C09106=1039.782,271.564,387.906,171.420,41.865,158.001
C09107=1039.788,271.812,387.876,171.423,41.867,158.001
C09108=1039.795,272.060,387.845,171.427,41.868,158.002
C09109=1039.802,272.308,387.814,171.430,41.870,158.002
C09110=1039.809,272.556,387.784,171.433,41.871,158.003
C09111=1039.815,272.805,387.753,171.437,41.873,158.003
C09112=1039.821,273.052,387.722,171.439,41.875,158.004
C09113=1039.828,273.300,387.692,171.443,41.876,158.004
C09114=1039.835,273.548,387.660,171.447,41.878,158.005
C09115=1039.842,273.796,387.630,171.449,41.880,158.006
C09116=1039.849,274.044,387.599,171.453,41.881,158.006
C09117=1039.855,274.292,387.568,171.457,41.883,158.007
C09118=1039.862,274.540,387.538,171.459,41.885,158.007
C09119=1039.869,274.788,387.507,171.463,41.887,158.008
C09120=1039.876,275.036,387.475,171.466,41.888,158.009
C09121=1039.882,275.285,387.445,171.469,41.890,158.009
C09122=1039.889,275.532,387.414,171.473,41.892,158.010
C09123=1039.895,275.780,387.383,171.475,41.893,158.010
C09124=1039.902,276.028,387.352,171.479,41.895,158.011
C09125=1039.908,276.276,387.321,171.483,41.897,158.011
C09126=1039.916,276.524,387.290,171.485,41.898,158.012
C09127=1039.925,276.838,387.251,171.490,41.901,158.013
C09128=1039.933,277.151,387.212,171.494,41.903,158.013
C09129=1039.942,277.465,387.173,171.498,41.905,158.014
C09130=1039.950,277.778,387.133,171.503,41.907,158.015
C09131=1039.957,278.027,387.103,171.507,41.909,158.016
C09132=1039.963,278.274,387.072,171.509,41.910,158.016
C09133=1039.970,278.522,387.040,171.513,41.912,158.017
C09134=1039.977,278.770,387.010,171.516,41.914,158.017
C09135=1039.983,279.018,386.979,171.519,41.916,158.018
C09136=1039.990,279.266,386.947,171.523,41.917,158.018
C09137=1039.997,279.514,386.916,171.527,41.919,158.019
C09138=1040.004,279.762,386.884,171.529,41.921,158.020
C09139=1040.010,280.010,386.854,171.533,41.923,158.020
C09140=1040.017,280.258,386.822,171.537,41.925,158.021
C09141=1040.023,280.506,386.791,171.539,41.926,158.021
C09142=1040.030,280.754,386.759,171.543,41.928,158.022
C09143=1040.037,281.002,386.728,171.547,41.930,158.023
C09144=1040.044,281.250,386.696,171.551,41.932,158.023
C09145=1040.050,281.498,386.665,171.553,41.933,158.024
C09146=1040.057,281.745,386.634,171.557,41.935,158.025
C09147=1040.063,281.993,386.602,171.561,41.937,158.025
C09148=1040.070,282.241,386.571,171.563,41.939,158.026
C09149=1040.077,282.489,386.540,171.567,41.941,158.026
C09150=1040.083,282.736,386.508,171.571,41.942,158.027
C09151=1040.090,282.984,386.477,171.574,41.944,158.028
C09152=1040.097,283.232,386.445,171.577,41.946,158.028
C09153=1040.104,283.481,386.413,171.581,41.948,158.029
C09154=1040.111,283.729,386.382,171.585,41.950,158.029
C09155=1040.118,283.977,386.351,171.588,41.951,158.030
C09156=1040.124,284.225,386.319,171.592,41.953,158.031
C09157=1040.131,284.473,386.288,171.595,41.954,158.031
C09158=1040.138,284.720,386.256,171.598,41.956,158.032
C09159=1040.145,284.968,386.225,171.602,41.958,158.033
C09160=1040.151,285.216,386.193,171.606,41.960,158.033
C09161=1040.158,285.463,386.161,171.608,41.962,158.034
C09162=1040.165,285.711,386.130,171.612,41.964,158.034
C09163=1040.172,285.959,386.098,171.616,41.965,158.035
C09164=1040.178,286.207,386.067,171.620,41.967,158.036
C09165=1040.185,286.455,386.036,171.623,41.969,158.036
C09166=1040.193,286.704,386.004,171.626,41.971,158.037
C09167=1040.200,286.951,385.972,171.630,41.973,158.037
C09168=1040.206,287.199,385.940,171.633,41.974,158.038
C09169=1040.212,287.447,385.908,171.637,41.976,158.039
C09170=1040.219,287.694,385.876,171.641,41.978,158.039
C09171=1040.226,287.942,385.845,171.645,41.980,158.040
C09172=1040.232,288.191,385.813,171.647,41.982,158.041
C09173=1040.239,288.438,385.780,171.651,41.984,158.041
C09174=1040.246,288.686,385.749,171.655,41.986,158.042
C09175=1040.253,288.934,385.717,171.659,41.988,158.043
C09176=1040.260,289.182,385.685,171.662,41.989,158.043
C09177=1040.266,289.430,385.653,171.665,41.991,158.044
C09178=1040.273,289.677,385.621,171.669,41.993,158.044
C09179=1040.280,289.925,385.589,171.673,41.995,158.045
C09180=1040.287,290.173,385.556,171.676,41.997,158.046
C09181=1040.293,290.421,385.525,171.680,41.999,158.046
C09182=1040.301,290.668,385.493,171.684,42.001,158.047
C09183=1040.309,290.994,385.451,171.688,42.003,158.048
C09184=1040.318,291.320,385.408,171.693,42.006,158.049
C09185=1040.327,291.645,385.366,171.698,42.008,158.050
C09186=1040.336,291.971,385.325,171.703,42.011,158.051
C09187=1040.343,292.218,385.292,171.707,42.013,158.051
C09188=1040.349,292.466,385.260,171.710,42.015,158.052
C09189=1040.356,292.714,385.228,171.713,42.017,158.052
C09190=1040.364,292.962,385.196,171.717,42.019,158.053
C09191=1040.370,293.209,385.163,171.721,42.021,158.054
C09192=1040.377,293.457,385.132,171.725,42.023,158.055
C09193=1040.384,293.704,385.099,171.728,42.025,158.055
C09194=1040.391,293.953,385.066,171.732,42.027,158.056
C09195=1040.397,294.201,385.035,171.736,42.029,158.057
C09196=1040.404,294.448,385.002,171.740,42.031,158.057
C09197=1040.411,294.696,384.970,171.743,42.032,158.058
C09198=1040.418,294.944,384.937,171.747,42.034,158.058
C09199=1040.425,295.191,384.905,171.750,42.036,158.059
C09200=1040.431,295.439,384.873,171.754,42.038,158.060
C09201=1040.438,295.687,384.840,171.757,42.040,158.061
C09202=1040.445,295.935,384.807,171.761,42.043,158.061
C09203=1040.451,296.182,384.775,171.765,42.045,158.062
C09204=1040.458,296.431,384.742,171.769,42.047,158.063
C09205=1040.465,296.678,384.709,171.773,42.048,158.063
C09206=1040.471,296.926,384.677,171.777,42.050,158.064
C09207=1040.477,297.173,384.644,171.780,42.052,158.065
C09208=1040.484,297.422,384.611,171.784,42.054,158.065
C09209=1040.491,297.669,384.578,171.788,42.057,158.066
C09210=1040.498,297.916,384.546,171.792,42.059,158.067
C09211=1040.505,298.165,384.513,171.795,42.061,158.068
C09212=1040.511,298.412,384.480,171.799,42.063,158.068
C09213=1040.517,298.660,384.447,171.802,42.065,158.069
C09214=1040.525,298.907,384.414,171.806,42.067,158.070
C09215=1040.531,299.155,384.381,171.810,42.070,158.071
C09216=1040.538,299.402,384.349,171.814,42.072,158.071
C09217=1040.545,299.651,384.315,171.818,42.074,158.072
C09218=1040.551,299.898,384.283,171.822,42.076,158.073
C09219=1040.558,300.146,384.250,171.825,42.077,158.073
C09220=1040.565,300.394,384.217,171.829,42.080,158.074
C09221=1040.571,300.641,384.184,171.833,42.082,158.075
C09222=1040.578,300.889,384.151,171.837,42.084,158.075
C09223=1040.585,301.136,384.119,171.841,42.086,158.076
C09224=1040.592,301.385,384.086,171.845,42.088,158.077
C09225=1040.599,301.632,384.052,171.849,42.091,158.078
C09226=1040.606,301.880,384.019,171.852,42.092,158.078
C09227=1040.612,302.128,383.986,171.856,42.094,158.079
C09228=1040.620,302.375,383.953,171.860,42.096,158.080
C09229=1040.626,302.623,383.920,171.864,42.099,158.081
C09230=1040.633,302.871,383.887,171.868,42.101,158.081
C09231=1040.640,303.118,383.854,171.872,42.103,158.082
C09232=1040.647,303.366,383.821,171.876,42.106,158.083
C09233=1040.653,303.614,383.788,171.879,42.107,158.083
C09234=1040.661,303.861,383.755,171.883,42.109,158.084
C09235=1040.667,304.109,383.722,171.887,42.111,158.085
C09236=1040.674,304.356,383.688,171.891,42.114,158.086
C09237=1040.681,304.604,383.655,171.896,42.116,158.086
C09238=1040.687,304.852,383.622,171.900,42.118,158.087
C09239=1040.697,305.194,383.576,171.905,42.121,158.088
C09240=1040.707,305.536,383.530,171.910,42.124,158.089
C09241=1040.717,305.878,383.485,171.915,42.127,158.090
C09242=1040.726,306.220,383.439,171.921,42.130,158.091
C09243=1040.733,306.467,383.406,171.925,42.132,158.092
C09244=1040.740,306.715,383.372,171.929,42.134,158.093
C09245=1040.747,306.963,383.339,171.933,42.137,158.094
C09246=1040.754,307.210,383.305,171.937,42.139,158.094
C09247=1040.761,307.458,383.272,171.941,42.141,158.095
C09248=1040.769,307.705,383.239,171.945,42.143,158.096
C09249=1040.775,307.953,383.206,171.950,42.145,158.097
C09250=1040.782,308.201,383.172,171.954,42.148,158.097
C09251=1040.789,308.448,383.138,171.957,42.150,158.098
C09252=1040.796,308.695,383.105,171.961,42.151,158.099
C09253=1040.803,308.944,383.072,171.965,42.154,158.100
C09254=1040.810,309.191,383.038,171.969,42.156,158.100
C09255=1040.818,309.439,383.005,171.973,42.159,158.101
C09256=1040.824,309.686,382.972,171.978,42.160,158.102
C09257=1040.831,309.934,382.938,171.982,42.163,158.103
C09258=1040.839,310.182,382.904,171.986,42.165,158.103
C09259=1040.846,310.429,382.871,171.990,42.167,158.104
C09260=1040.852,310.676,382.837,171.993,42.169,158.105
C09261=1040.859,310.925,382.804,171.998,42.172,158.106
C09262=1040.867,311.172,382.770,172.002,42.174,158.106
C09263=1040.874,311.420,382.737,172.006,42.176,158.107
C09264=1040.882,311.667,382.703,172.010,42.178,158.108
C09265=1040.889,311.915,382.669,172.014,42.181,158.109
C09266=1040.895,312.162,382.636,172.019,42.183,158.110
C09267=1040.903,312.410,382.602,172.023,42.185,158.110
C09268=1040.909,312.658,382.568,172.027,42.188,158.111
C09269=1040.916,312.905,382.534,172.031,42.190,158.112
C09270=1040.922,313.152,382.500,172.035,42.192,158.113
C09271=1040.929,313.400,382.466,172.039,42.195,158.114
C09272=1040.936,313.648,382.431,172.044,42.197,158.115
C09273=1040.943,313.895,382.397,172.048,42.200,158.115
C09274=1040.949,314.142,382.363,172.051,42.202,158.116
C09275=1040.956,314.390,382.329,172.055,42.204,158.117
C09276=1040.964,314.638,382.295,172.060,42.207,158.118
C09277=1040.970,314.885,382.260,172.064,42.209,158.119
C09278=1040.978,315.133,382.226,172.069,42.212,158.119
C09279=1040.984,315.381,382.192,172.073,42.214,158.120
C09280=1040.991,315.627,382.158,172.077,42.217,158.121
C09281=1040.997,315.875,382.123,172.080,42.219,158.122
C09282=1041.005,316.123,382.089,172.085,42.221,158.123
C09283=1041.011,316.370,382.054,172.089,42.224,158.124
C09284=1041.019,316.618,382.020,172.093,42.226,158.124
C09285=1041.025,316.866,381.986,172.097,42.229,158.125
C09286=1041.033,317.113,381.952,172.101,42.231,158.126
C09287=1041.039,317.361,381.917,172.106,42.234,158.127
C09288=1041.046,317.609,381.883,172.110,42.236,158.128
C09289=1041.052,317.855,381.849,172.114,42.239,158.129
C09290=1041.060,318.103,381.815,172.119,42.241,158.130
C09291=1041.066,318.350,381.780,172.123,42.244,158.130
C09292=1041.074,318.598,381.746,172.127,42.246,158.131
C09293=1041.080,318.845,381.711,172.132,42.249,158.132
C09294=1041.088,319.093,381.677,172.137,42.251,158.133
C09295=1041.098,319.440,381.628,172.142,42.255,158.134
C09296=1041.107,319.787,381.580,172.148,42.258,158.135
C09297=1041.117,320.133,381.531,172.155,42.261,158.137
C09298=1041.127,320.480,381.483,172.160,42.265,158.138
C09299=1041.134,320.728,381.448,172.164,42.268,158.139
C09300=1041.141,320.975,381.414,172.169,42.270,158.139
C09301=1041.148,321.222,381.378,172.173,42.273,158.140
C09302=1041.155,321.470,381.345,172.177,42.275,158.141
C09303=1041.162,321.717,381.310,172.182,42.277,158.142
C09304=1041.169,321.964,381.275,172.186,42.280,158.143
C09305=1041.177,322.213,381.240,172.191,42.282,158.144
C09306=1041.184,322.460,381.206,172.195,42.285,158.145
C09307=1041.191,322.707,381.171,172.200,42.288,158.146
C09308=1041.198,322.954,381.136,172.205,42.290,158.147
C09309=1041.205,323.202,381.102,172.209,42.293,158.147
C09310=1041.212,323.449,381.067,172.213,42.295,158.148
C09311=1041.220,323.697,381.032,172.218,42.298,158.149
C09312=1041.226,323.945,380.996,172.222,42.300,158.150
C09313=1041.234,324.192,380.962,172.227,42.303,158.151
C09314=1041.241,324.439,380.927,172.231,42.306,158.152
C09315=1041.248,324.686,380.892,172.235,42.308,158.153
C09316=1041.255,324.935,380.857,172.240,42.311,158.154
C09317=1041.263,325.182,380.823,172.244,42.313,158.154
C09318=1041.270,325.429,380.788,172.249,42.316,158.155
C09319=1041.277,325.676,380.753,172.253,42.319,158.156
C09320=1041.284,325.925,380.718,172.257,42.321,158.157
C09321=1041.291,326.172,380.683,172.262,42.324,158.158
C09322=1041.299,326.419,380.648,172.266,42.327,158.159
C09323=1041.306,326.667,380.612,172.272,42.329,158.160
C09324=1041.314,326.914,380.578,172.276,42.332,158.161
C09325=1041.320,327.161,380.543,172.281,42.334,158.162
C09326=1041.328,327.409,380.508,172.285,42.337,158.163
C09327=1041.336,327.656,380.472,172.290,42.339,158.164
C09328=1041.342,327.903,380.437,172.294,42.342,158.164
C09329=1041.350,328.151,380.402,172.299,42.345,158.165
C09330=1041.357,328.398,380.367,172.303,42.347,158.166
C09331=1041.365,328.646,380.332,172.308,42.350,158.167
C09332=1041.372,328.894,380.297,172.312,42.353,158.168
C09333=1041.379,329.140,380.261,172.317,42.355,158.169
C09334=1041.386,329.388,380.225,172.322,42.358,158.170
C09335=1041.393,329.636,380.190,172.327,42.361,158.171
C09336=1041.400,329.882,380.154,172.331,42.364,158.172
C09337=1041.408,330.131,380.119,172.336,42.367,158.173
C09338=1041.414,330.378,380.084,172.340,42.369,158.174
C09339=1041.422,330.625,380.048,172.345,42.372,158.175
C09340=1041.429,330.873,380.013,172.349,42.375,158.176
C09341=1041.436,331.119,379.977,172.355,42.378,158.177
C09342=1041.443,331.368,379.941,172.359,42.381,158.178
C09343=1041.450,331.614,379.905,172.364,42.383,158.179
C09344=1041.458,331.862,379.870,172.368,42.386,158.180
C09345=1041.465,332.109,379.834,172.373,42.389,158.181
C09346=1041.472,332.357,379.798,172.377,42.392,158.182
C09347=1041.479,332.604,379.763,172.383,42.395,158.183
C09348=1041.487,332.852,379.727,172.387,42.398,158.184
C09349=1041.494,333.099,379.691,172.392,42.400,158.185
C09350=1041.501,333.345,379.655,172.396,42.403,158.186
C09351=1041.511,333.688,379.606,172.403,42.407,158.187
C09352=1041.521,334.030,379.556,172.409,42.411,158.188
C09353=1041.531,334.371,379.507,172.416,42.415,158.190
C09354=1041.542,334.714,379.457,172.423,42.419,158.191
C09355=1041.548,334.961,379.422,172.428,42.422,158.192
C09356=1041.556,335.208,379.386,172.432,42.425,158.193
C09357=1041.564,335.456,379.349,172.437,42.428,158.194
C09358=1041.571,335.703,379.313,172.442,42.431,158.195
C09359=1041.578,335.950,379.277,172.447,42.433,158.196
C09360=1041.585,336.197,379.241,172.452,42.436,158.197
C09361=1041.592,336.445,379.205,172.456,42.439,158.198
C09362=1041.599,336.692,379.169,172.461,42.442,158.199
C09363=1041.607,336.939,379.133,172.467,42.445,158.200
C09364=1041.614,337.187,379.096,172.471,42.448,158.201
C09365=1041.621,337.434,379.061,172.476,42.451,158.202
C09366=1041.629,337.681,379.024,172.480,42.454,158.203
C09367=1041.635,337.929,378.988,172.486,42.457,158.204
C09368=1041.643,338.176,378.952,172.491,42.461,158.206
C09369=1041.651,338.423,378.915,172.495,42.464,158.207
C09370=1041.658,338.670,378.879,172.501,42.467,158.208
C09371=1041.665,338.917,378.842,172.506,42.470,158.209
C09372=1041.672,339.165,378.806,172.510,42.473,158.210
C09373=1041.680,339.412,378.770,172.515,42.476,158.211
C09374=1041.687,339.659,378.734,172.521,42.479,158.212
C09375=1041.694,339.907,378.697,172.525,42.482,158.213
C09376=1041.702,340.153,378.660,172.530,42.485,158.214
C09377=1041.710,340.401,378.624,172.536,42.488,158.215
C09378=1041.717,340.649,378.587,172.540,42.491,158.216
C09379=1041.724,340.895,378.551,172.545,42.494,158.217
C09380=1041.732,341.142,378.514,172.550,42.497,158.218
C09381=1041.738,341.390,378.477,172.556,42.500,158.219
C09382=1041.746,341.637,378.441,172.560,42.503,158.220
C09383=1041.754,341.884,378.404,172.565,42.506,158.221
C09384=1041.760,342.131,378.368,172.571,42.509,158.222
C09385=1041.768,342.379,378.332,172.576,42.513,158.224
C09386=1041.775,342.626,378.294,172.580,42.516,158.225
C09387=1041.783,342.873,378.258,172.586,42.519,158.226
C09388=1041.790,343.120,378.220,172.591,42.522,158.227
C09389=1041.798,343.368,378.184,172.596,42.525,158.228
C09390=1041.805,343.614,378.147,172.601,42.529,158.229
C09391=1041.812,343.862,378.111,172.606,42.532,158.230
C09392=1041.820,344.109,378.073,172.611,42.535,158.231
C09393=1041.827,344.356,378.036,172.617,42.538,158.232
C09394=1041.834,344.603,378.000,172.621,42.542,158.234
C09395=1041.842,344.851,377.962,172.626,42.545,158.235
C09396=1041.850,345.097,377.925,172.632,42.548,158.236
C09397=1041.857,345.345,377.888,172.637,42.551,158.237
C09398=1041.865,345.592,377.851,172.643,42.555,158.238
C09399=1041.872,345.839,377.814,172.647,42.558,158.239
C09400=1041.879,346.086,377.776,172.652,42.561,158.240
C09401=1041.887,346.334,377.740,172.658,42.564,158.241
C09402=1041.893,346.580,377.703,172.663,42.567,158.243
C09403=1041.901,346.827,377.665,172.669,42.571,158.244
C09404=1041.909,347.074,377.628,172.673,42.574,158.245
C09405=1041.916,347.321,377.591,172.678,42.578,158.246
C09406=1041.924,347.569,377.553,172.684,42.581,158.247
C09407=1041.934,347.907,377.503,172.691,42.585,158.249
C09408=1041.944,348.246,377.452,172.699,42.590,158.250
C09409=1041.954,348.583,377.401,172.705,42.594,158.252
C09410=1041.965,348.922,377.350,172.713,42.599,158.254
C09411=1041.972,349.169,377.312,172.718,42.602,158.255
C09412=1041.980,349.416,377.275,172.723,42.606,158.256
C09413=1041.988,349.664,377.237,172.729,42.609,158.257
C09414=1041.995,349.910,377.199,172.734,42.613,158.258
C09415=1042.003,350.157,377.162,172.740,42.616,158.260
C09416=1042.010,350.404,377.125,172.745,42.620,158.261
C09417=1042.018,350.651,377.087,172.751,42.623,158.262
C09418=1042.025,350.899,377.050,172.756,42.627,158.263
C09419=1042.032,351.145,377.011,172.762,42.630,158.264
C09420=1042.040,351.392,376.974,172.767,42.633,158.266
C09421=1042.048,351.640,376.936,172.772,42.637,158.267
C09422=1042.055,351.887,376.898,172.777,42.641,158.268
C09423=1042.062,352.134,376.860,172.783,42.644,158.269
C09424=1042.070,352.381,376.823,172.788,42.647,158.270
C09425=1042.078,352.627,376.785,172.794,42.651,158.272
C09426=1042.086,352.875,376.747,172.799,42.654,158.273
C09427=1042.093,353.122,376.710,172.805,42.658,158.274
C09428=1042.100,353.369,376.671,172.810,42.661,158.275
C09429=1042.108,353.616,376.634,172.816,42.665,158.277
C09430=1042.116,353.863,376.595,172.821,42.669,158.278
C09431=1042.123,354.110,376.558,172.827,42.672,158.279
C09432=1042.131,354.357,376.519,172.832,42.676,158.280
C09433=1042.139,354.604,376.482,172.838,42.679,158.282
C09434=1042.146,354.851,376.443,172.843,42.683,158.283
C09435=1042.154,355.097,376.405,172.849,42.687,158.284
C09436=1042.161,355.345,376.367,172.854,42.690,158.285
C09437=1042.169,355.592,376.329,172.860,42.694,158.287
C09438=1042.177,355.838,376.291,172.866,42.698,158.288
C09439=1042.185,356.086,376.253,172.872,42.701,158.289
C09440=1042.193,356.332,376.215,172.878,42.704,158.290
C09441=1042.200,356.579,376.177,172.883,42.708,158.292
C09442=1042.208,356.826,376.138,172.889,42.712,158.293
C09443=1042.215,357.074,376.100,172.894,42.716,158.294
C09444=1042.223,357.321,376.062,172.900,42.719,158.296
C09445=1042.231,357.567,376.023,172.906,42.723,158.297
C09446=1042.239,357.814,375.985,172.911,42.727,158.298
C09447=1042.246,358.061,375.946,172.917,42.731,158.300
C09448=1042.254,358.307,375.908,172.922,42.734,158.301
C09449=1042.262,358.555,375.870,172.928,42.738,158.302
C09450=1042.269,358.802,375.831,172.934,42.742,158.303
C09451=1042.277,359.049,375.792,172.940,42.745,158.305
C09452=1042.285,359.295,375.754,172.946,42.749,158.306
C09453=1042.293,359.542,375.715,172.952,42.753,158.307
C09454=1042.300,359.789,375.677,172.957,42.757,158.309
C09455=1042.308,360.036,375.638,172.963,42.761,158.310
C09456=1042.316,360.283,375.600,172.968,42.764,158.311
C09457=1042.323,360.530,375.561,172.975,42.768,158.313
C09458=1042.332,360.777,375.522,172.981,42.772,158.314
C09459=1042.339,361.023,375.483,172.986,42.776,158.315
C09460=1042.347,361.271,375.445,172.992,42.780,158.317
C09461=1042.354,361.517,375.406,172.998,42.784,158.318
C09462=1042.363,361.764,375.367,173.005,42.787,158.320
C09463=1042.373,362.108,375.313,173.012,42.793,158.322
C09464=1042.385,362.453,375.259,173.020,42.799,158.323
C09465=1042.395,362.797,375.204,173.029,42.804,158.325
C09466=1042.406,363.140,375.149,173.037,42.809,158.327
C09467=1042.414,363.388,375.111,173.043,42.813,158.329
C09468=1042.422,363.634,375.071,173.049,42.817,158.330
C09469=1042.429,363.881,375.033,173.055,42.821,158.331
C09470=1042.437,364.128,374.993,173.061,42.826,158.333
C09471=1042.445,364.374,374.953,173.067,42.830,158.334
C09472=1042.453,364.621,374.915,173.073,42.834,158.336
C09473=1042.461,364.868,374.875,173.079,42.838,158.337
C09474=1042.469,365.115,374.837,173.085,42.842,158.339
C09475=1042.476,365.362,374.797,173.091,42.846,158.340
C09476=1042.484,365.608,374.758,173.098,42.850,158.342
C09477=1042.492,365.855,374.718,173.104,42.854,158.343
C09478=1042.500,366.102,374.679,173.109,42.858,158.344
C09479=1042.508,366.349,374.639,173.116,42.862,158.346
C09480=1042.516,366.596,374.600,173.122,42.866,158.347
C09481=1042.524,366.842,374.560,173.128,42.870,158.349
C09482=1042.532,367.088,374.521,173.134,42.874,158.350
C09483=1042.540,367.335,374.481,173.140,42.879,158.352
C09484=1042.548,367.582,374.442,173.146,42.883,158.353
C09485=1042.556,367.829,374.403,173.153,42.886,158.355
C09486=1042.564,368.076,374.363,173.159,42.891,158.356
C09487=1042.572,368.323,374.323,173.165,42.895,158.357
C09488=1042.580,368.569,374.284,173.172,42.899,158.359
C09489=1042.588,368.816,374.244,173.177,42.903,158.360
C09490=1042.597,369.062,374.204,173.184,42.908,158.362
C09491=1042.604,369.309,374.165,173.190,42.912,158.363
C09492=1042.612,369.555,374.125,173.197,42.916,158.365
C09493=1042.620,369.802,374.085,173.203,42.920,158.366
C09494=1042.628,370.049,374.045,173.209,42.924,158.368
C09495=1042.636,370.296,374.006,173.216,42.929,158.370
C09496=1042.644,370.543,373.966,173.221,42.933,158.371
C09497=1042.653,370.789,373.926,173.228,42.937,158.373
C09498=1042.661,371.036,373.886,173.234,42.942,158.374
C09499=1042.669,371.283,373.846,173.241,42.946,158.376
C09500=1042.677,371.529,373.805,173.247,42.951,158.377
C09501=1042.684,371.776,373.765,173.254,42.954,158.379
C09502=1042.692,372.022,373.725,173.260,42.959,158.380
C09503=1042.701,372.269,373.685,173.267,42.963,158.382
C09504=1042.709,372.515,373.645,173.273,42.968,158.383
C09505=1042.717,372.762,373.605,173.280,42.972,158.385
C09506=1042.725,373.008,373.564,173.286,42.977,158.387
C09507=1042.732,373.255,373.524,173.293,42.981,158.388
C09508=1042.740,373.502,373.484,173.299,42.986,158.390
C09509=1042.749,373.748,373.444,173.306,42.990,158.391
C09510=1042.757,373.995,373.404,173.312,42.994,158.393
C09511=1042.766,374.242,373.363,173.319,42.999,158.394
C09512=1042.774,374.488,373.322,173.325,43.003,158.396
C09513=1042.781,374.735,373.282,173.332,43.008,158.398
C09514=1042.789,374.981,373.242,173.339,43.013,158.399
C09515=1042.797,375.227,373.201,173.345,43.017,158.401
C09516=1042.806,375.474,373.160,173.352,43.021,158.403
C09517=1042.815,375.720,373.120,173.358,43.026,158.404
C09518=1042.822,375.967,373.080,173.365,43.031,158.406
C09519=1042.834,376.331,373.019,173.375,43.037,158.408
C09520=1042.847,376.695,372.960,173.385,43.044,158.411
C09521=1042.859,377.058,372.899,173.395,43.051,158.413
C09522=1042.871,377.422,372.840,173.404,43.058,158.416
C09523=1042.880,377.669,372.799,173.411,43.062,158.417
C09524=1042.888,377.915,372.758,173.419,43.067,158.419
C09525=1042.897,378.162,372.717,173.425,43.072,158.421
C09526=1042.905,378.409,372.676,173.432,43.077,158.422
C09527=1042.913,378.655,372.636,173.439,43.081,158.424
C09528=1042.922,378.901,372.594,173.446,43.086,158.426
C09529=1042.930,379.148,372.553,173.452,43.090,158.427
C09530=1042.938,379.394,372.512,173.459,43.095,158.429
C09531=1042.947,379.640,372.471,173.466,43.100,158.431
C09532=1042.955,379.887,372.430,173.474,43.105,158.433
C09533=1042.963,380.134,372.389,173.480,43.109,158.434
C09534=1042.972,380.380,372.347,173.487,43.114,158.436
C09535=1042.980,380.626,372.307,173.494,43.119,158.438
C09536=1042.987,380.872,372.265,173.501,43.124,158.439
C09537=1042.996,381.119,372.224,173.508,43.129,158.441
C09538=1043.004,381.365,372.182,173.515,43.134,158.443
C09539=1043.013,381.611,372.141,173.522,43.139,158.445
C09540=1043.022,381.858,372.100,173.529,43.144,158.446
C09541=1043.029,382.104,372.058,173.537,43.149,158.448
C09542=1043.038,382.351,372.017,173.543,43.154,158.450
C09543=1043.046,382.597,371.975,173.550,43.158,158.452
C09544=1043.055,382.843,371.934,173.557,43.163,158.454
C09545=1043.063,383.089,371.892,173.565,43.168,158.455
C09546=1043.071,383.336,371.851,173.572,43.173,158.457
C09547=1043.080,383.583,371.809,173.579,43.178,158.459
C09548=1043.089,383.828,371.768,173.586,43.183,158.461
C09549=1043.097,384.075,371.725,173.593,43.188,158.463
C09550=1043.106,384.321,371.683,173.600,43.193,158.464
C09551=1043.115,384.568,371.642,173.607,43.198,158.466
C09552=1043.123,384.813,371.600,173.615,43.204,158.468
C09553=1043.131,385.060,371.558,173.622,43.208,158.470
C09554=1043.140,385.306,371.516,173.629,43.213,158.472
C09555=1043.149,385.553,371.475,173.637,43.219,158.474
C09556=1043.157,385.799,371.433,173.644,43.223,158.475
C09557=1043.166,386.045,371.391,173.651,43.229,158.477
C09558=1043.175,386.292,371.349,173.659,43.234,158.479
C09559=1043.184,386.538,371.308,173.666,43.239,158.481
C09560=1043.192,386.785,371.265,173.673,43.244,158.483
C09561=1043.201,387.030,371.223,173.681,43.249,158.485
C09562=1043.209,387.276,371.181,173.688,43.254,158.487
C09563=1043.218,387.523,371.139,173.696,43.260,158.488
C09564=1043.226,387.769,371.097,173.703,43.264,158.490
C09565=1043.236,388.015,371.055,173.710,43.270,158.492
C09566=1043.245,388.261,371.013,173.718,43.275,158.494
C09567=1043.253,388.508,370.971,173.725,43.281,158.496
C09568=1043.262,388.754,370.929,173.733,43.285,158.498
C09569=1043.270,389.000,370.886,173.740,43.291,158.500
C09570=1043.279,389.246,370.843,173.749,43.296,158.502
C09571=1043.288,389.492,370.801,173.756,43.301,158.504
C09572=1043.296,389.739,370.758,173.764,43.307,158.506
C09573=1043.305,389.984,370.716,173.771,43.312,158.508
C09574=1043.314,390.231,370.674,173.779,43.318,158.510
C09575=1043.328,390.628,370.604,173.791,43.326,158.513
C09576=1043.342,391.025,370.536,173.804,43.335,158.516
C09577=1043.356,391.423,370.467,173.816,43.344,158.519
C09578=1043.371,391.821,370.398,173.828,43.353,158.523
C09579=1043.380,392.067,370.356,173.837,43.358,158.525
C09580=1043.388,392.313,370.313,173.845,43.364,158.527
C09581=1043.397,392.559,370.270,173.852,43.369,158.529
C09582=1043.405,392.805,370.226,173.860,43.375,158.531
C09583=1043.415,393.051,370.184,173.867,43.380,158.533
C09584=1043.424,393.297,370.140,173.876,43.386,158.535
C09585=1043.432,393.543,370.097,173.884,43.391,158.537
C09586=1043.442,393.789,370.054,173.891,43.397,158.539
C09587=1043.450,394.035,370.011,173.900,43.403,158.541
C09588=1043.459,394.282,369.968,173.908,43.408,158.543
C09589=1043.468,394.528,369.925,173.915,43.414,158.545
C09590=1043.477,394.773,369.882,173.924,43.419,158.547
C09591=1043.486,395.020,369.838,173.932,43.425,158.549
C09592=1043.495,395.266,369.795,173.939,43.431,158.551
C09593=1043.504,395.511,369.752,173.948,43.437,158.554
C09594=1043.514,395.757,369.709,173.956,43.443,158.556
C09595=1043.522,396.003,369.665,173.964,43.448,158.558
C09596=1043.531,396.249,369.622,173.972,43.454,158.560
C09597=1043.540,396.495,369.578,173.980,43.460,158.562
C09598=1043.549,396.741,369.535,173.988,43.466,158.564
C09599=1043.558,396.987,369.491,173.997,43.471,158.566
C09600=1043.567,397.233,369.447,174.005,43.478,158.569
C09601=1043.576,397.479,369.404,174.013,43.484,158.571
C09602=1043.585,397.725,369.360,174.021,43.489,158.573
C09603=1043.594,397.970,369.316,174.030,43.495,158.575
C09604=1043.603,398.216,369.272,174.038,43.501,158.577
C09605=1043.612,398.463,369.229,174.047,43.507,158.580
C09606=1043.621,398.709,369.185,174.055,43.513,158.582
C09607=1043.631,398.955,369.141,174.063,43.519,158.584
C09608=1043.639,399.200,369.097,174.071,43.525,158.586
C09609=1043.649,399.446,369.054,174.080,43.531,158.589
C09610=1043.659,399.692,369.010,174.088,43.537,158.591
C09611=1043.668,399.938,368.966,174.097,43.543,158.593
C09612=1043.677,400.184,368.922,174.105,43.549,158.595
C09613=1043.686,400.430,368.878,174.114,43.555,158.598
C09614=1043.695,400.676,368.833,174.122,43.561,158.600
C09615=1043.704,400.922,368.789,174.131,43.567,158.602
C09616=1043.713,401.168,368.745,174.140,43.573,158.604
C09617=1043.723,401.413,368.700,174.148,43.580,158.607
C09618=1043.732,401.659,368.657,174.157,43.585,158.609
C09619=1043.741,401.905,368.612,174.166,43.592,158.611
C09620=1043.751,402.150,368.568,174.174,43.598,158.614
C09621=1043.760,402.397,368.523,174.183,43.604,158.616
C09622=1043.769,402.643,368.479,174.192,43.610,158.618
C09623=1043.778,402.888,368.434,174.200,43.617,158.621
C09624=1043.788,403.134,368.390,174.209,43.623,158.623
C09625=1043.797,403.379,368.345,174.218,43.629,158.625
C09626=1043.806,403.626,368.301,174.226,43.636,158.628
C09627=1043.816,403.871,368.256,174.235,43.642,158.630
C09628=1043.825,404.117,368.211,174.244,43.648,158.632
C09629=1043.834,404.363,368.166,174.254,43.655,158.635
C09630=1043.844,404.609,368.121,174.262,43.661,158.637
C09631=1043.851,404.817,368.083,174.269,43.666,158.639
C09632=1043.860,405.026,368.045,174.277,43.672,158.641
C09633=1043.867,405.234,368.007,174.285,43.677,158.643
C09634=1043.876,405.442,367.969,174.293,43.683,158.646
C09635=1043.883,405.651,367.931,174.300,43.688,158.648
C09636=1043.891,405.859,367.892,174.308,43.694,158.650
C09637=1043.899,406.067,367.855,174.316,43.699,158.652
C09638=1043.908,406.276,367.816,174.324,43.705,158.654
C09639=1043.917,406.522,367.771,174.333,43.711,158.656
C09640=1043.926,406.768,367.726,174.342,43.718,158.659
C09641=1043.936,407.013,367.681,174.351,43.725,158.661
C09642=1043.945,407.259,367.635,174.360,43.731,158.664
C09643=1043.955,407.504,367.591,174.369,43.738,158.666
C09644=1043.965,407.750,367.545,174.378,43.745,158.669
C09645=1043.974,407.996,367.499,174.387,43.751,158.671
C09646=1043.984,408.241,367.454,174.397,43.758,158.674
C09647=1043.993,408.487,367.409,174.406,43.765,158.677
C09648=1044.004,408.733,367.363,174.415,43.771,158.679
C09649=1044.013,408.979,367.318,174.425,43.778,158.682
C09650=1044.023,409.223,367.272,174.434,43.785,158.684
C09651=1044.032,409.470,367.226,174.443,43.791,158.687
C09652=1044.042,409.715,367.181,174.454,43.798,158.689
C09653=1044.053,409.961,367.136,174.463,43.805,158.692
C09654=1044.062,410.206,367.090,174.473,43.812,158.695
C09655=1044.072,410.452,367.045,174.482,43.818,158.697
C09656=1044.081,410.698,366.998,174.492,43.826,158.700
C09657=1044.092,410.943,366.953,174.501,43.832,158.703
C09658=1044.101,411.189,366.907,174.510,43.839,158.705
C09659=1044.112,411.435,366.861,174.521,43.846,158.708
C09660=1044.121,411.680,366.815,174.531,43.853,158.711
C09661=1044.132,411.926,366.769,174.540,43.860,158.713
C09662=1044.141,412.171,366.724,174.550,43.867,158.716
C09663=1044.151,412.417,366.678,174.559,43.874,158.719
C09664=1044.161,412.662,366.632,174.570,43.881,158.721
C09665=1044.170,412.908,366.585,174.579,43.888,158.724
C09666=1044.181,413.153,366.538,174.589,43.895,158.727
C09667=1044.190,413.399,366.492,174.599,43.902,158.729
C09668=1044.200,413.644,366.446,174.609,43.909,158.732
C09669=1044.210,413.890,366.399,174.619,43.916,158.735
C09670=1044.220,414.135,366.353,174.629,43.924,158.738
C09671=1044.230,414.381,366.306,174.639,43.931,158.741
C09672=1044.240,414.626,366.259,174.649,43.938,158.743
C09673=1044.250,414.872,366.213,174.660,43.945,158.746
C09674=1044.260,415.117,366.167,174.669,43.952,158.749
C09675=1044.270,415.363,366.120,174.679,43.960,158.752
C09676=1044.280,415.608,366.073,174.690,43.967,158.755
C09677=1044.290,415.854,366.026,174.700,43.975,158.758
C09678=1044.301,416.099,365.980,174.710,43.982,158.760
C09679=1044.311,416.345,365.933,174.720,43.989,158.763
C09680=1044.321,416.590,365.886,174.731,43.996,158.766
C09681=1044.331,416.835,365.839,174.741,44.004,158.769
C09682=1044.341,417.080,365.792,174.752,44.011,158.772
C09683=1044.351,417.326,365.746,174.762,44.019,158.775
C09684=1044.362,417.571,365.699,174.772,44.026,158.778
C09685=1044.372,417.817,365.651,174.783,44.033,158.781
C09686=1044.382,418.062,365.604,174.793,44.041,158.784
C09687=1044.393,418.307,365.557,174.804,44.049,158.787
C09688=1044.403,418.552,365.510,174.815,44.056,158.790
C09689=1044.413,418.798,365.462,174.825,44.064,158.793
C09690=1044.423,419.043,365.415,174.836,44.071,158.795
C09691=1044.432,419.270,365.371,174.846,44.078,158.798
C09692=1044.442,419.496,365.328,174.855,44.085,158.801
C09693=1044.451,419.723,365.284,174.866,44.092,158.804
C09694=1044.462,419.949,365.240,174.876,44.100,158.807
C09695=1044.471,420.176,365.196,174.886,44.107,158.810
C09696=1044.480,420.402,365.152,174.896,44.114,158.812
C09697=1044.490,420.628,365.108,174.906,44.121,158.815
C09698=1044.499,420.855,365.064,174.916,44.129,158.818
C09699=1044.510,421.099,365.016,174.927,44.136,158.821
C09700=1044.521,421.345,364.968,174.938,44.144,158.824
C09701=1044.531,421.590,364.920,174.949,44.152,158.827
C09702=1044.541,421.835,364.873,174.960,44.159,158.830
C09703=1044.552,422.081,364.825,174.971,44.167,158.834
C09704=1044.563,422.325,364.777,174.982,44.175,158.837
C09705=1044.572,422.571,364.729,174.993,44.183,158.840
C09706=1044.583,422.816,364.681,175.005,44.191,158.843
C09707=1044.594,423.061,364.633,175.016,44.199,158.846
C09708=1044.605,423.306,364.584,175.027,44.208,158.850
C09709=1044.615,423.551,364.537,175.039,44.215,158.853
C09710=1044.627,423.796,364.488,175.050,44.223,158.856
C09711=1044.638,424.042,364.440,175.061,44.231,158.859
C09712=1044.647,424.287,364.391,175.073,44.240,158.862
C09713=1044.659,424.532,364.343,175.085,44.247,158.866
C09714=1044.670,424.778,364.295,175.096,44.256,158.869
C09715=1044.680,425.022,364.247,175.108,44.264,158.872
C09716=1044.691,425.267,364.197,175.119,44.272,158.876
C09717=1044.702,425.513,364.149,175.131,44.281,158.879
C09718=1044.712,425.758,364.100,175.142,44.289,158.882
C09719=1044.723,426.002,364.051,175.154,44.297,158.886
C09720=1044.734,426.248,364.003,175.166,44.305,158.889
C09721=1044.744,426.492,363.954,175.178,44.314,158.892
C09722=1044.755,426.737,363.906,175.189,44.322,158.896
C09723=1044.767,426.982,363.857,175.202,44.330,158.899
C09724=1044.777,427.227,363.807,175.213,44.339,158.903
C09725=1044.789,427.473,363.759,175.225,44.347,158.906
C09726=1044.799,427.718,363.709,175.238,44.356,158.909
C09727=1044.810,427.962,363.660,175.249,44.364,158.913
C09728=1044.821,428.206,363.611,175.262,44.373,158.916
C09729=1044.832,428.451,363.562,175.274,44.381,158.920
C09730=1044.843,428.696,363.513,175.286,44.390,158.923
C09731=1044.854,428.941,363.463,175.298,44.398,158.927
C09732=1044.866,429.186,363.414,175.311,44.407,158.930
C09733=1044.876,429.431,363.365,175.323,44.416,158.934
C09734=1044.887,429.676,363.315,175.335,44.424,158.937
C09735=1044.898,429.907,363.268,175.347,44.433,158.941
C09736=1044.908,430.137,363.222,175.359,44.441,158.944
C09737=1044.919,430.368,363.175,175.370,44.449,158.948
C09738=1044.930,430.599,363.128,175.382,44.458,158.951
C09739=1044.940,430.829,363.081,175.394,44.466,158.955
C09740=1044.950,431.060,363.034,175.406,44.474,158.958
C09741=1044.961,431.290,362.986,175.418,44.482,158.961
C09742=1044.971,431.521,362.940,175.429,44.491,158.965
C09743=1044.983,431.766,362.890,175.442,44.500,158.969
C09744=1044.994,432.010,362.840,175.455,44.508,158.972
C09745=1045.005,432.255,362.790,175.468,44.517,158.976
C09746=1045.016,432.499,362.739,175.481,44.526,158.980
C09747=1045.028,432.745,362.690,175.493,44.535,158.983
C09748=1045.039,432.989,362.640,175.507,44.545,158.987
C09749=1045.051,433.234,362.589,175.520,44.554,158.991
C09750=1045.063,433.478,362.539,175.533,44.562,158.995
C09751=1045.073,433.702,362.493,175.545,44.571,158.998
C09752=1045.084,433.924,362.447,175.557,44.579,159.002
C09753=1045.094,434.147,362.401,175.569,44.587,159.005
C09754=1045.104,434.370,362.355,175.581,44.596,159.009
C09755=1045.115,434.593,362.310,175.594,44.604,159.012
C09756=1045.126,434.816,362.263,175.605,44.613,159.016
C09757=1045.136,435.039,362.217,175.617,44.621,159.019
C09758=1045.147,435.262,362.170,175.630,44.630,159.023
C09759=1045.159,435.506,362.120,175.643,44.639,159.027
C09760=1045.170,435.751,362.070,175.657,44.648,159.031
C09761=1045.182,435.995,362.019,175.670,44.657,159.034
C09762=1045.194,436.240,361.967,175.684,44.667,159.038
C09763=1045.205,436.484,361.917,175.698,44.676,159.042
C09764=1045.217,436.729,361.865,175.711,44.686,159.046
C09765=1045.230,436.973,361.815,175.725,44.695,159.051
C09766=1045.242,437.217,361.763,175.739,44.705,159.055
C09767=1045.253,437.462,361.712,175.753,44.714,159.059
C09768=1045.265,437.707,361.661,175.766,44.724,159.063
C09769=1045.277,437.952,361.610,175.781,44.734,159.067
C09770=1045.288,438.195,361.558,175.795,44.743,159.071
C09771=1045.300,438.439,361.507,175.809,44.753,159.075
C09772=1045.312,438.684,361.455,175.823,44.762,159.079
C09773=1045.324,438.928,361.404,175.838,44.772,159.083
C09774=1045.336,439.172,361.352,175.852,44.782,159.088
C09775=1045.348,439.417,361.300,175.866,44.792,159.092
C09776=1045.360,439.661,361.249,175.880,44.802,159.096
C09777=1045.373,439.906,361.196,175.895,44.811,159.100
C09778=1045.385,440.150,361.145,175.910,44.821,159.104
C09779=1045.397,440.394,361.093,175.923,44.831,159.109
C09780=1045.409,440.638,361.041,175.938,44.841,159.113
C09781=1045.421,440.883,360.989,175.953,44.851,159.117
C09782=1045.433,441.126,360.937,175.968,44.861,159.122
C09783=1045.446,441.371,360.885,175.983,44.871,159.126
C09784=1045.458,441.615,360.833,175.997,44.881,159.130
C09785=1045.470,441.859,360.780,176.012,44.891,159.135
C09786=1045.482,442.104,360.727,176.027,44.902,159.139
C09787=1045.495,442.348,360.675,176.042,44.911,159.143
C09788=1045.507,442.592,360.623,176.057,44.922,159.148
C09789=1045.520,442.836,360.571,176.073,44.932,159.152
C09790=1045.532,443.079,360.518,176.088,44.942,159.157
C09791=1045.545,443.324,360.465,176.103,44.953,159.161
C09792=1045.556,443.568,360.413,176.118,44.963,159.166
C09793=1045.569,443.812,360.359,176.133,44.973,159.170
C09794=1045.582,444.056,360.307,176.149,44.984,159.175
C09795=1045.595,444.300,360.254,176.165,44.994,159.180
C09796=1045.607,444.545,360.202,176.181,45.005,159.184
C09797=1045.620,444.788,360.149,176.196,45.015,159.189
C09798=1045.633,445.032,360.096,176.211,45.025,159.193
C09799=1045.645,445.275,360.043,176.228,45.036,159.198
C09800=1045.658,445.518,359.990,176.243,45.046,159.203
C09801=1045.671,445.761,359.938,176.258,45.057,159.207
C09802=1045.686,446.005,359.885,176.275,45.067,159.212
C09803=1045.701,446.248,359.835,176.291,45.077,159.217
C09804=1045.716,446.491,359.784,176.307,45.087,159.221
C09805=1045.732,446.736,359.734,176.323,45.096,159.226
C09806=1045.749,446.980,359.684,176.340,45.106,159.230
C09807=1045.766,447.223,359.634,176.356,45.116,159.235
C09808=1045.785,447.468,359.586,176.372,45.125,159.239
C09809=1045.804,447.712,359.537,176.389,45.135,159.244
C09810=1045.823,447.957,359.489,176.405,45.144,159.248
C09811=1045.845,448.224,359.438,176.424,45.154,159.253
C09812=1045.868,448.490,359.387,176.441,45.164,159.257
C09813=1045.891,448.757,359.336,176.460,45.174,159.262
C09814=1045.915,449.025,359.286,176.478,45.183,159.267
C09815=1045.937,449.270,359.242,176.496,45.191,159.271
C09816=1045.961,449.515,359.196,176.512,45.200,159.275
C09817=1045.985,449.760,359.153,176.529,45.208,159.280
C09818=1046.011,450.005,359.109,176.547,45.216,159.284
C09819=1046.035,450.250,359.066,176.563,45.224,159.288
C09820=1046.062,450.496,359.024,176.581,45.233,159.292
C09821=1046.088,450.742,358.982,176.599,45.241,159.297
C09822=1046.116,450.987,358.939,176.616,45.248,159.301
C09823=1045.810,451.023,358.632,176.618,45.333,159.326
C09824=1045.782,450.778,358.672,176.601,45.325,159.322
C09825=1045.755,450.533,358.714,176.583,45.317,159.317
C09826=1045.729,450.287,358.758,176.565,45.309,159.313
C09827=1045.704,450.041,358.800,176.548,45.302,159.309
C09828=1045.679,449.796,358.844,176.531,45.293,159.305
C09829=1045.654,449.551,358.888,176.514,45.285,159.301
C09830=1045.631,449.306,358.933,176.496,45.276,159.296
C09831=1045.608,449.061,358.977,176.479,45.268,159.292
C09832=1045.585,448.811,359.024,176.462,45.259,159.288
C09833=1045.562,448.561,359.071,176.445,45.250,159.283
C09834=1045.541,448.309,359.119,176.428,45.242,159.279
C09835=1045.520,448.060,359.167,176.411,45.232,159.274
C09836=1045.501,447.815,359.214,176.394,45.223,159.270
C09837=1045.482,447.571,359.263,176.377,45.214,159.265
C09838=1045.463,447.327,359.311,176.361,45.205,159.261
C09839=1045.445,447.083,359.360,176.344,45.195,159.257
C09840=1045.428,446.839,359.409,176.328,45.185,159.252
C09841=1045.411,446.595,359.459,176.312,45.176,159.247
C09842=1045.396,446.351,359.510,176.295,45.166,159.243
C09843=1045.380,446.108,359.561,176.279,45.156,159.238
C09844=1045.365,445.864,359.613,176.263,45.146,159.234
C09845=1045.351,445.620,359.665,176.248,45.136,159.229
C09846=1045.338,445.377,359.717,176.231,45.126,159.225
C09847=1045.325,445.134,359.770,176.216,45.115,159.220
C09848=1045.313,444.891,359.823,176.199,45.105,159.215
C09849=1045.300,444.647,359.876,176.184,45.094,159.211
C09850=1045.287,444.402,359.929,176.168,45.084,159.206
C09851=1045.275,444.159,359.982,176.153,45.074,159.201
C09852=1045.262,443.915,360.035,176.137,45.064,159.197
C09853=1045.249,443.670,360.087,176.121,45.053,159.192
C09854=1045.236,443.427,360.140,176.106,45.043,159.188
C09855=1045.224,443.182,360.193,176.091,45.033,159.183
C09856=1045.212,442.938,360.245,176.076,45.022,159.179
C09857=1045.199,442.694,360.299,176.061,45.012,159.174
C09858=1045.187,442.451,360.351,176.045,45.002,159.170
C09859=1045.174,442.206,360.403,176.030,44.992,159.165
C09860=1045.162,441.962,360.455,176.015,44.982,159.161
C09861=1045.150,441.718,360.507,176.000,44.972,159.157
C09862=1045.138,441.473,360.560,175.985,44.962,159.152
C09863=1045.126,441.229,360.613,175.970,44.952,159.148
C09864=1045.113,440.986,360.665,175.955,44.942,159.144
C09865=1045.101,440.740,360.716,175.940,44.932,159.139
C09866=1045.089,440.496,360.769,175.926,44.922,159.135
C09867=1045.076,440.253,360.821,175.911,44.912,159.131
C09868=1045.065,440.008,360.872,175.897,44.902,159.126
C09869=1045.052,439.764,360.924,175.883,44.892,159.122
C09870=1045.041,439.520,360.976,175.868,44.883,159.118
C09871=1045.028,439.275,361.028,175.853,44.873,159.114
C09872=1045.016,439.031,361.080,175.839,44.863,159.109
C09873=1045.004,438.787,361.132,175.825,44.854,159.105
C09874=1044.992,438.542,361.183,175.811,44.844,159.101
C09875=1044.980,438.298,361.234,175.796,44.835,159.097
C09876=1044.968,438.053,361.286,175.783,44.825,159.093
C09877=1044.957,437.809,361.337,175.768,44.816,159.089
C09878=1044.945,437.565,361.388,175.754,44.806,159.085
C09879=1044.932,437.321,361.439,175.740,44.797,159.081
C09880=1044.920,437.076,361.491,175.726,44.787,159.077
C09881=1044.908,436.832,361.542,175.713,44.778,159.073
C09882=1044.897,436.587,361.593,175.698,44.768,159.068
C09883=1044.885,436.342,361.644,175.685,44.759,159.064
C09884=1044.874,436.098,361.695,175.671,44.749,159.060
C09885=1044.862,435.854,361.746,175.657,44.740,159.057
C09886=1044.850,435.608,361.797,175.643,44.731,159.052
C09887=1044.838,435.364,361.848,175.630,44.722,159.049
C09888=1044.827,435.141,361.894,175.617,44.713,159.045
C09889=1044.817,434.917,361.941,175.606,44.705,159.042
C09890=1044.806,434.694,361.987,175.594,44.696,159.038
C09891=1044.795,434.470,362.033,175.581,44.688,159.034
C09892=1044.784,434.246,362.079,175.569,44.680,159.031
C09893=1044.774,434.022,362.126,175.556,44.672,159.027
C09894=1044.763,433.798,362.172,175.545,44.663,159.024
C09895=1044.753,433.574,362.217,175.533,44.655,159.020
C09896=1044.742,433.330,362.267,175.520,44.646,159.017
C09897=1044.730,433.085,362.317,175.506,44.637,159.013
C09898=1044.719,432.841,362.368,175.493,44.628,159.009
C09899=1044.707,432.596,362.418,175.480,44.619,159.005
C09900=1044.695,432.352,362.468,175.467,44.610,159.002
C09901=1044.684,432.107,362.519,175.454,44.601,158.998
C09902=1044.673,431.862,362.569,175.441,44.592,158.994
C09903=1044.661,431.617,362.618,175.429,44.583,158.990
C09904=1044.650,431.373,362.669,175.416,44.574,158.987
C09905=1044.639,431.128,362.719,175.403,44.566,158.983
C09906=1044.627,430.883,362.768,175.390,44.557,158.979
C09907=1044.616,430.638,362.819,175.378,44.548,158.976
C09908=1044.605,430.394,362.868,175.365,44.540,158.972
C09909=1044.594,430.149,362.918,175.352,44.531,158.969
C09910=1044.583,429.904,362.968,175.340,44.522,158.965
C09911=1044.572,429.660,363.017,175.328,44.514,158.961
C09912=1044.561,429.414,363.066,175.315,44.505,158.958
C09913=1044.550,429.170,363.116,175.303,44.496,158.954
C09914=1044.539,428.925,363.165,175.290,44.488,158.951
C09915=1044.528,428.680,363.215,175.278,44.479,158.947
C09916=1044.517,428.435,363.264,175.266,44.471,158.944
C09917=1044.506,428.190,363.314,175.254,44.462,158.940
C09918=1044.495,427.946,363.363,175.241,44.454,158.937
C09919=1044.483,427.701,363.412,175.230,44.446,158.933
C09920=1044.473,427.455,363.461,175.217,44.437,158.930
C09921=1044.462,427.211,363.510,175.205,44.428,158.926
C09922=1044.450,426.966,363.559,175.194,44.420,158.923
C09923=1044.440,426.720,363.608,175.181,44.412,158.920
C09924=1044.429,426.475,363.657,175.169,44.404,158.916
C09925=1044.418,426.231,363.705,175.158,44.395,158.913
C09926=1044.407,425.986,363.754,175.146,44.387,158.910
C09927=1044.396,425.741,363.803,175.134,44.379,158.906
C09928=1044.386,425.495,363.852,175.122,44.371,158.903
C09929=1044.375,425.251,363.900,175.111,44.362,158.899
C09930=1044.364,425.006,363.949,175.099,44.355,158.896
C09931=1044.353,424.760,363.998,175.087,44.346,158.893
C09932=1044.343,424.516,364.046,175.076,44.338,158.890
C09933=1044.332,424.270,364.094,175.064,44.330,158.886
C09934=1044.321,424.025,364.142,175.053,44.322,158.883
C09935=1044.310,423.780,364.190,175.042,44.314,158.880
C09936=1044.300,423.534,364.239,175.030,44.306,158.877
C09937=1044.289,423.290,364.287,175.018,44.299,158.873
C09938=1044.278,423.044,364.335,175.006,44.290,158.870
C09939=1044.268,422.800,364.383,174.995,44.282,158.867
C09940=1044.256,422.547,364.433,174.984,44.274,158.864
C09941=1044.246,422.293,364.483,174.972,44.266,158.860
C09942=1044.235,422.040,364.532,174.961,44.258,158.857
C09943=1044.223,421.787,364.582,174.950,44.250,158.854
C09944=1044.213,421.541,364.630,174.939,44.242,158.851
C09945=1044.203,421.296,364.678,174.927,44.234,158.848
C09946=1044.193,421.051,364.725,174.916,44.227,158.845
C09947=1044.182,420.805,364.773,174.905,44.219,158.841
C09948=1044.173,420.597,364.814,174.896,44.212,158.839
C09949=1044.164,420.387,364.854,174.886,44.206,158.836
C09950=1044.155,420.178,364.895,174.877,44.199,158.834
C09951=1044.147,419.969,364.936,174.868,44.192,158.831
C09952=1044.137,419.759,364.977,174.859,44.186,158.828
C09953=1044.128,419.550,365.017,174.849,44.179,158.826
C09954=1044.120,419.340,365.057,174.840,44.173,158.823
C09955=1044.111,419.131,365.099,174.831,44.167,158.821
C09956=1044.101,418.886,365.146,174.820,44.159,158.818
C09957=1044.091,418.641,365.193,174.809,44.151,158.815
C09958=1044.081,418.396,365.240,174.798,44.144,158.812
C09959=1044.070,418.150,365.287,174.788,44.136,158.809
C09960=1044.060,417.905,365.335,174.777,44.129,158.806
C09961=1044.049,417.659,365.382,174.767,44.122,158.803
C09962=1044.038,417.414,365.429,174.757,44.114,158.800
C09963=1044.028,417.169,365.476,174.746,44.107,158.797
C09964=1044.018,416.923,365.523,174.736,44.100,158.794
C09965=1044.008,416.678,365.570,174.725,44.092,158.791
C09966=1043.997,416.433,365.616,174.715,44.084,158.788
C09967=1043.987,416.187,365.663,174.704,44.078,158.785
C09968=1043.978,415.942,365.710,174.693,44.070,158.782
C09969=1043.968,415.697,365.757,174.684,44.063,158.780
C09970=1043.958,415.451,365.804,174.673,44.056,158.777
C09971=1043.948,415.206,365.851,174.663,44.048,158.774
C09972=1043.937,414.960,365.897,174.653,44.041,158.771
C09973=1043.927,414.714,365.943,174.643,44.034,158.768
C09974=1043.917,414.470,365.990,174.633,44.027,158.766
C09975=1043.908,414.224,366.036,174.622,44.020,158.763
C09976=1043.897,413.979,366.083,174.613,44.013,158.760
C09977=1043.887,413.733,366.130,174.603,44.006,158.757
C09978=1043.877,413.488,366.176,174.592,43.999,158.754
C09979=1043.868,413.242,366.222,174.583,43.992,158.752
C09980=1043.858,412.996,366.269,174.573,43.984,158.749
C09981=1043.848,412.751,366.314,174.562,43.977,158.746
C09982=1043.838,412.505,366.361,174.553,43.970,158.743
C09983=1043.828,412.260,366.408,174.543,43.963,158.741
C09984=1043.819,412.014,366.453,174.534,43.956,158.738
C09985=1043.808,411.768,366.499,174.523,43.949,158.735
C09986=1043.799,411.523,366.545,174.514,43.943,158.733
C09987=1043.788,411.277,366.591,174.504,43.936,158.730
C09988=1043.778,411.031,366.637,174.495,43.929,158.727
C09989=1043.768,410.786,366.683,174.484,43.922,158.725
C09990=1043.758,410.540,366.729,174.475,43.915,158.722
C09991=1043.749,410.295,366.774,174.465,43.909,158.719
C09992=1043.738,410.049,366.820,174.456,43.902,158.717
C09993=1043.729,409.804,366.866,174.446,43.895,158.714
C09994=1043.719,409.558,366.911,174.437,43.888,158.712
C09995=1043.709,409.312,366.957,174.427,43.881,158.709
C09996=1043.700,409.067,367.002,174.418,43.875,158.706
//INST
///DATE 2021/06/25 14:48
///ATTR SC,RW,RJ
////FRAME ROBOT
///GROUP1 RB1
NOP
MOVL C00000 V=800.0 PL=0
MOVL C00001 V=800.0 PL=0
MOVL C00002 V=800.0 PL=0
MOVL C00003 V=800.0 PL=0
MOVL C00004 V=800.0 PL=0
MOVL C00005 V=800.0 PL=0
MOVL C00006 V=800.0 PL=0
MOVL C00007 V=800.0 PL=0
MOVL C00008 V=800.0 PL=0
MOVL C00009 V=800.0 PL=0
MOVL C00010 V=800.0 PL=0
MOVL C00011 V=800.0 PL=0
MOVL C00012 V=800.0 PL=0
MOVL C00013 V=800.0 PL=0
MOVL C00014 V=800.0 PL=0
MOVL C00015 V=800.0 PL=0
MOVL C00016 V=800.0 PL=0
MOVL C00017 V=800.0 PL=0
MOVL C00018 V=800.0 PL=0
MOVL C00019 V=800.0 PL=0
MOVL C00020 V=800.0 PL=0
MOVL C00021 V=800.0 PL=0
MOVL C00022 V=800.0 PL=0
MOVL C00023 V=800.0 PL=0
MOVL C00024 V=800.0 PL=0
MOVL C00025 V=800.0 PL=0
MOVL C00026 V=800.0 PL=0
MOVL C00027 V=800.0 PL=0
MOVL C00028 V=800.0 PL=0
MOVL C00029 V=800.0 PL=0
MOVL C00030 V=800.0 PL=0
MOVL C00031 V=800.0 PL=0
MOVL C00032 V=800.0 PL=0
MOVL C00033 V=800.0 PL=0
MOVL C00034 V=800.0 PL=0
MOVL C00035 V=800.0 PL=0
MOVL C00036 V=800.0 PL=0
MOVL C00037 V=800.0 PL=0
MOVL C00038 V=800.0 PL=0
MOVL C00039 V=800.0 PL=0
MOVL C00040 V=800.0 PL=0
MOVL C00041 V=800.0 PL=0
MOVL C00042 V=800.0 PL=0
MOVL C00043 V=800.0 PL=0
MOVL C00044 V=800.0 PL=0
MOVL C00045 V=800.0 PL=0
MOVL C00046 V=800.0 PL=0
MOVL C00047 V=800.0 PL=0
MOVL C00048 V=800.0 PL=0
MOVL C00049 V=800.0 PL=0
MOVL C00050 V=800.0 PL=0
MOVL C00051 V=800.0 PL=0
MOVL C00052 V=800.0 PL=0
MOVL C00053 V=800.0 PL=0
MOVL C00054 V=800.0 PL=0
MOVL C00055 V=800.0 PL=0
MOVL C00056 V=800.0 PL=0
MOVL C00057 V=800.0 PL=0
MOVL C00058 V=800.0 PL=0
MOVL C00059 V=800.0 PL=0
MOVL C00060 V=800.0 PL=0
MOVL C00061 V=800.0 PL=0
MOVL C00062 V=800.0 PL=0
MOVL C00063 V=800.0 PL=0
MOVL C00064 V=800.0 PL=0
MOVL C00065 V=800.0 PL=0
MOVL C00066 V=800.0 PL=0
MOVL C00067 V=800.0 PL=0
MOVL C00068 V=800.0 PL=0
MOVL C00069 V=800.0 PL=0
MOVL C00070 V=800.0 PL=0
MOVL C00071 V=800.0 PL=0
MOVL C00072 V=800.0 PL=0
MOVL C00073 V=800.0 PL=0
MOVL C00074 V=800.0 PL=0
MOVL C00075 V=800.0 PL=0
MOVL C00076 V=800.0 PL=0
MOVL C00077 V=800.0 PL=0
MOVL C00078 V=800.0 PL=0
MOVL C00079 V=800.0 PL=0
MOVL C00080 V=800.0 PL=0
MOVL C00081 V=800.0 PL=0
MOVL C00082 V=800.0 PL=0
MOVL C00083 V=800.0 PL=0
MOVL C00084 V=800.0 PL=0
MOVL C00085 V=800.0 PL=0
MOVL C00086 V=800.0 PL=0
MOVL C00087 V=800.0 PL=0
MOVL C00088 V=800.0 PL=0
MOVL C00089 V=800.0 PL=0
MOVL C00090 V=800.0 PL=0
MOVL C00091 V=800.0 PL=0
MOVL C00092 V=800.0 PL=0
MOVL C00093 V=800.0 PL=0
MOVL C00094 V=800.0 PL=0
MOVL C00095 V=800.0 PL=0
MOVL C00096 V=800.0 PL=0
MOVL C00097 V=800.0 PL=0
MOVL C00098 V=800.0 PL=0
MOVL C00099 V=800.0 PL=0
MOVL C00100 V=800.0 PL=0
MOVL C00101 V=800.0 PL=0
MOVL C00102 V=800.0 PL=0
MOVL C00103 V=800.0 PL=0
MOVL C00104 V=800.0 PL=0
MOVL C00105 V=800.0 PL=0
MOVL C00106 V=800.0 PL=0
MOVL C00107 V=800.0 PL=0
MOVL C00108 V=800.0 PL=0
MOVL C00109 V=800.0 PL=0
MOVL C00110 V=800.0 PL=0
MOVL C00111 V=800.0 PL=0
MOVL C00112 V=800.0 PL=0
MOVL C00113 V=800.0 PL=0
MOVL C00114 V=800.0 PL=0
MOVL C00115 V=800.0 PL=0
MOVL C00116 V=800.0 PL=0
MOVL C00117 V=800.0 PL=0
MOVL C00118 V=800.0 PL=0
MOVL C00119 V=800.0 PL=0
MOVL C00120 V=800.0 PL=0
MOVL C00121 V=800.0 PL=0
MOVL C00122 V=800.0 PL=0
MOVL C00123 V=800.0 PL=0
MOVL C00124 V=800.0 PL=0
MOVL C00125 V=800.0 PL=0
MOVL C00126 V=800.0 PL=0
MOVL C00127 V=800.0 PL=0
MOVL C00128 V=800.0 PL=0
MOVL C00129 V=800.0 PL=0
MOVL C00130 V=800.0 PL=0
MOVL C00131 V=800.0 PL=0
MOVL C00132 V=800.0 PL=0
MOVL C00133 V=800.0 PL=0
MOVL C00134 V=800.0 PL=0
MOVL C00135 V=800.0 PL=0
MOVL C00136 V=800.0 PL=0
MOVL C00137 V=800.0 PL=0
MOVL C00138 V=800.0 PL=0
MOVL C00139 V=800.0 PL=0
MOVL C00140 V=800.0 PL=0
MOVL C00141 V=800.0 PL=0
MOVL C00142 V=800.0 PL=0
MOVL C00143 V=800.0 PL=0
MOVL C00144 V=800.0 PL=0
MOVL C00145 V=800.0 PL=0
MOVL C00146 V=800.0 PL=0
MOVL C00147 V=800.0 PL=0
MOVL C00148 V=800.0 PL=0
MOVL C00149 V=800.0 PL=0
MOVL C00150 V=800.0 PL=0
MOVL C00151 V=800.0 PL=0
MOVL C00152 V=800.0 PL=0
MOVL C00153 V=800.0 PL=0
MOVL C00154 V=800.0 PL=0
MOVL C00155 V=800.0 PL=0
MOVL C00156 V=800.0 PL=0
MOVL C00157 V=800.0 PL=0
MOVL C00158 V=800.0 PL=0
MOVL C00159 V=800.0 PL=0
MOVL C00160 V=800.0 PL=0
MOVL C00161 V=800.0 PL=0
MOVL C00162 V=800.0 PL=0
MOVL C00163 V=800.0 PL=0
MOVL C00164 V=800.0 PL=0
MOVL C00165 V=800.0 PL=0
MOVL C00166 V=800.0 PL=0
MOVL C00167 V=800.0 PL=0
MOVL C00168 V=800.0 PL=0
MOVL C00169 V=800.0 PL=0
MOVL C00170 V=800.0 PL=0
MOVL C00171 V=800.0 PL=0
MOVL C00172 V=800.0 PL=0
MOVL C00173 V=800.0 PL=0
MOVL C00174 V=800.0 PL=0
MOVL C00175 V=800.0 PL=0
MOVL C00176 V=800.0 PL=0
MOVL C00177 V=800.0 PL=0
MOVL C00178 V=800.0 PL=0
MOVL C00179 V=800.0 PL=0
MOVL C00180 V=800.0 PL=0
MOVL C00181 V=800.0 PL=0
MOVL C00182 V=800.0 PL=0
MOVL C00183 V=800.0 PL=0
MOVL C00184 V=800.0 PL=0
MOVL C00185 V=800.0 PL=0
MOVL C00186 V=800.0 PL=0
MOVL C00187 V=800.0 PL=0
MOVL C00188 V=800.0 PL=0
MOVL C00189 V=800.0 PL=0
MOVL C00190 V=800.0 PL=0
MOVL C00191 V=800.0 PL=0
MOVL C00192 V=800.0 PL=0
MOVL C00193 V=800.0 PL=0
MOVL C00194 V=800.0 PL=0
MOVL C00195 V=800.0 PL=0
MOVL C00196 V=800.0 PL=0
MOVL C00197 V=800.0 PL=0
MOVL C00198 V=800.0 PL=0
MOVL C00199 V=800.0 PL=0
MOVL C00200 V=800.0 PL=0
MOVL C00201 V=800.0 PL=0
MOVL C00202 V=800.0 PL=0
MOVL C00203 V=800.0 PL=0
MOVL C00204 V=800.0 PL=0
MOVL C00205 V=800.0 PL=0
MOVL C00206 V=800.0 PL=0
MOVL C00207 V=800.0 PL=0
MOVL C00208 V=800.0 PL=0
MOVL C00209 V=800.0 PL=0
MOVL C00210 V=800.0 PL=0
MOVL C00211 V=800.0 PL=0
MOVL C00212 V=800.0 PL=0
MOVL C00213 V=800.0 PL=0
MOVL C00214 V=800.0 PL=0
MOVL C00215 V=800.0 PL=0
MOVL C00216 V=800.0 PL=0
MOVL C00217 V=800.0 PL=0
MOVL C00218 V=800.0 PL=0
MOVL C00219 V=800.0 PL=0
MOVL C00220 V=800.0 PL=0
MOVL C00221 V=800.0 PL=0
MOVL C00222 V=800.0 PL=0
MOVL C00223 V=800.0 PL=0
MOVL C00224 V=800.0 PL=0
MOVL C00225 V=800.0 PL=0
MOVL C00226 V=800.0 PL=0
MOVL C00227 V=800.0 PL=0
MOVL C00228 V=800.0 PL=0
MOVL C00229 V=800.0 PL=0
MOVL C00230 V=800.0 PL=0
MOVL C00231 V=800.0 PL=0
MOVL C00232 V=800.0 PL=0
MOVL C00233 V=800.0 PL=0
MOVL C00234 V=800.0 PL=0
MOVL C00235 V=800.0 PL=0
MOVL C00236 V=800.0 PL=0
MOVL C00237 V=800.0 PL=0
MOVL C00238 V=800.0 PL=0
MOVL C00239 V=800.0 PL=0
MOVL C00240 V=800.0 PL=0
MOVL C00241 V=800.0 PL=0
MOVL C00242 V=800.0 PL=0
MOVL C00243 V=800.0 PL=0
MOVL C00244 V=800.0 PL=0
MOVL C00245 V=800.0 PL=0
MOVL C00246 V=800.0 PL=0
MOVL C00247 V=800.0 PL=0
MOVL C00248 V=800.0 PL=0
MOVL C00249 V=800.0 PL=0
MOVL C00250 V=800.0 PL=0
MOVL C00251 V=800.0 PL=0
MOVL C00252 V=800.0 PL=0
MOVL C00253 V=800.0 PL=0
MOVL C00254 V=800.0 PL=0
MOVL C00255 V=800.0 PL=0
MOVL C00256 V=800.0 PL=0
MOVL C00257 V=800.0 PL=0
MOVL C00258 V=800.0 PL=0
MOVL C00259 V=800.0 PL=0
MOVL C00260 V=800.0 PL=0
MOVL C00261 V=800.0 PL=0
MOVL C00262 V=800.0 PL=0
MOVL C00263 V=800.0 PL=0
MOVL C00264 V=800.0 PL=0
MOVL C00265 V=800.0 PL=0
MOVL C00266 V=800.0 PL=0
MOVL C00267 V=800.0 PL=0
MOVL C00268 V=800.0 PL=0
MOVL C00269 V=800.0 PL=0
MOVL C00270 V=800.0 PL=0
MOVL C00271 V=800.0 PL=0
MOVL C00272 V=800.0 PL=0
MOVL C00273 V=800.0 PL=0
MOVL C00274 V=800.0 PL=0
MOVL C00275 V=800.0 PL=0
MOVL C00276 V=800.0 PL=0
MOVL C00277 V=800.0 PL=0
MOVL C00278 V=800.0 PL=0
MOVL C00279 V=800.0 PL=0
MOVL C00280 V=800.0 PL=0
MOVL C00281 V=800.0 PL=0
MOVL C00282 V=800.0 PL=0
MOVL C00283 V=800.0 PL=0
MOVL C00284 V=800.0 PL=0
MOVL C00285 V=800.0 PL=0
MOVL C00286 V=800.0 PL=0
MOVL C00287 V=800.0 PL=0
MOVL C00288 V=800.0 PL=0
MOVL C00289 V=800.0 PL=0
MOVL C00290 V=800.0 PL=0
MOVL C00291 V=800.0 PL=0
MOVL C00292 V=800.0 PL=0
MOVL C00293 V=800.0 PL=0
MOVL C00294 V=800.0 PL=0
MOVL C00295 V=800.0 PL=0
MOVL C00296 V=800.0 PL=0
MOVL C00297 V=800.0 PL=0
MOVL C00298 V=800.0 PL=0
MOVL C00299 V=800.0 PL=0
MOVL C00300 V=800.0 PL=0
MOVL C00301 V=800.0 PL=0
MOVL C00302 V=800.0 PL=0
MOVL C00303 V=800.0 PL=0
MOVL C00304 V=800.0 PL=0
MOVL C00305 V=800.0 PL=0
MOVL C00306 V=800.0 PL=0
MOVL C00307 V=800.0 PL=0
MOVL C00308 V=800.0 PL=0
MOVL C00309 V=800.0 PL=0
MOVL C00310 V=800.0 PL=0
MOVL C00311 V=800.0 PL=0
MOVL C00312 V=800.0 PL=0
MOVL C00313 V=800.0 PL=0
MOVL C00314 V=800.0 PL=0
MOVL C00315 V=800.0 PL=0
MOVL C00316 V=800.0 PL=0
MOVL C00317 V=800.0 PL=0
MOVL C00318 V=800.0 PL=0
MOVL C00319 V=800.0 PL=0
MOVL C00320 V=800.0 PL=0
MOVL C00321 V=800.0 PL=0
MOVL C00322 V=800.0 PL=0
MOVL C00323 V=800.0 PL=0
MOVL C00324 V=800.0 PL=0
MOVL C00325 V=800.0 PL=0
MOVL C00326 V=800.0 PL=0
MOVL C00327 V=800.0 PL=0
MOVL C00328 V=800.0 PL=0
MOVL C00329 V=800.0 PL=0
MOVL C00330 V=800.0 PL=0
MOVL C00331 V=800.0 PL=0
MOVL C00332 V=800.0 PL=0
MOVL C00333 V=800.0 PL=0
MOVL C00334 V=800.0 PL=0
MOVL C00335 V=800.0 PL=0
MOVL C00336 V=800.0 PL=0
MOVL C00337 V=800.0 PL=0
MOVL C00338 V=800.0 PL=0
MOVL C00339 V=800.0 PL=0
MOVL C00340 V=800.0 PL=0
MOVL C00341 V=800.0 PL=0
MOVL C00342 V=800.0 PL=0
MOVL C00343 V=800.0 PL=0
MOVL C00344 V=800.0 PL=0
MOVL C00345 V=800.0 PL=0
MOVL C00346 V=800.0 PL=0
MOVL C00347 V=800.0 PL=0
MOVL C00348 V=800.0 PL=0
MOVL C00349 V=800.0 PL=0
MOVL C00350 V=800.0 PL=0
MOVL C00351 V=800.0 PL=0
MOVL C00352 V=800.0 PL=0
MOVL C00353 V=800.0 PL=0
MOVL C00354 V=800.0 PL=0
MOVL C00355 V=800.0 PL=0
MOVL C00356 V=800.0 PL=0
MOVL C00357 V=800.0 PL=0
MOVL C00358 V=800.0 PL=0
MOVL C00359 V=800.0 PL=0
MOVL C00360 V=800.0 PL=0
MOVL C00361 V=800.0 PL=0
MOVL C00362 V=800.0 PL=0
MOVL C00363 V=800.0 PL=0
MOVL C00364 V=800.0 PL=0
MOVL C00365 V=800.0 PL=0
MOVL C00366 V=800.0 PL=0
MOVL C00367 V=800.0 PL=0
MOVL C00368 V=800.0 PL=0
MOVL C00369 V=800.0 PL=0
MOVL C00370 V=800.0 PL=0
MOVL C00371 V=800.0 PL=0
MOVL C00372 V=800.0 PL=0
MOVL C00373 V=800.0 PL=0
MOVL C00374 V=800.0 PL=0
MOVL C00375 V=800.0 PL=0
MOVL C00376 V=800.0 PL=0
MOVL C00377 V=800.0 PL=0
MOVL C00378 V=800.0 PL=0
MOVL C00379 V=800.0 PL=0
MOVL C00380 V=800.0 PL=0
MOVL C00381 V=800.0 PL=0
MOVL C00382 V=800.0 PL=0
MOVL C00383 V=800.0 PL=0
MOVL C00384 V=800.0 PL=0
MOVL C00385 V=800.0 PL=0
MOVL C00386 V=800.0 PL=0
MOVL C00387 V=800.0 PL=0
MOVL C00388 V=800.0 PL=0
MOVL C00389 V=800.0 PL=0
MOVL C00390 V=800.0 PL=0
MOVL C00391 V=800.0 PL=0
MOVL C00392 V=800.0 PL=0
MOVL C00393 V=800.0 PL=0
MOVL C00394 V=800.0 PL=0
MOVL C00395 V=800.0 PL=0
MOVL C00396 V=800.0 PL=0
MOVL C00397 V=800.0 PL=0
MOVL C00398 V=800.0 PL=0
MOVL C00399 V=800.0 PL=0
MOVL C00400 V=800.0 PL=0
MOVL C00401 V=800.0 PL=0
MOVL C00402 V=800.0 PL=0
MOVL C00403 V=800.0 PL=0
MOVL C00404 V=800.0 PL=0
MOVL C00405 V=800.0 PL=0
MOVL C00406 V=800.0 PL=0
MOVL C00407 V=800.0 PL=0
MOVL C00408 V=800.0 PL=0
MOVL C00409 V=800.0 PL=0
MOVL C00410 V=800.0 PL=0
MOVL C00411 V=800.0 PL=0
MOVL C00412 V=800.0 PL=0
MOVL C00413 V=800.0 PL=0
MOVL C00414 V=800.0 PL=0
MOVL C00415 V=800.0 PL=0
MOVL C00416 V=800.0 PL=0
MOVL C00417 V=800.0 PL=0
MOVL C00418 V=800.0 PL=0
MOVL C00419 V=800.0 PL=0
MOVL C00420 V=800.0 PL=0
MOVL C00421 V=800.0 PL=0
MOVL C00422 V=800.0 PL=0
MOVL C00423 V=800.0 PL=0
MOVL C00424 V=800.0 PL=0
MOVL C00425 V=800.0 PL=0
MOVL C00426 V=800.0 PL=0
MOVL C00427 V=800.0 PL=0
MOVL C00428 V=800.0 PL=0
MOVL C00429 V=800.0 PL=0
MOVL C00430 V=800.0 PL=0
MOVL C00431 V=800.0 PL=0
MOVL C00432 V=800.0 PL=0
MOVL C00433 V=800.0 PL=0
MOVL C00434 V=800.0 PL=0
MOVL C00435 V=800.0 PL=0
MOVL C00436 V=800.0 PL=0
MOVL C00437 V=800.0 PL=0
MOVL C00438 V=800.0 PL=0
MOVL C00439 V=800.0 PL=0
MOVL C00440 V=800.0 PL=0
MOVL C00441 V=800.0 PL=0
MOVL C00442 V=800.0 PL=0
MOVL C00443 V=800.0 PL=0
MOVL C00444 V=800.0 PL=0
MOVL C00445 V=800.0 PL=0
MOVL C00446 V=800.0 PL=0
MOVL C00447 V=800.0 PL=0
MOVL C00448 V=800.0 PL=0
MOVL C00449 V=800.0 PL=0
MOVL C00450 V=800.0 PL=0
MOVL C00451 V=800.0 PL=0
MOVL C00452 V=800.0 PL=0
MOVL C00453 V=800.0 PL=0
MOVL C00454 V=800.0 PL=0
MOVL C00455 V=800.0 PL=0
MOVL C00456 V=800.0 PL=0
MOVL C00457 V=800.0 PL=0
MOVL C00458 V=800.0 PL=0
MOVL C00459 V=800.0 PL=0
MOVL C00460 V=800.0 PL=0
MOVL C00461 V=800.0 PL=0
MOVL C00462 V=800.0 PL=0
MOVL C00463 V=800.0 PL=0
MOVL C00464 V=800.0 PL=0
MOVL C00465 V=800.0 PL=0
MOVL C00466 V=800.0 PL=0
MOVL C00467 V=800.0 PL=0
MOVL C00468 V=800.0 PL=0
MOVL C00469 V=800.0 PL=0
MOVL C00470 V=800.0 PL=0
MOVL C00471 V=800.0 PL=0
MOVL C00472 V=800.0 PL=0
MOVL C00473 V=800.0 PL=0
MOVL C00474 V=800.0 PL=0
MOVL C00475 V=800.0 PL=0
MOVL C00476 V=800.0 PL=0
MOVL C00477 V=800.0 PL=0
MOVL C00478 V=800.0 PL=0
MOVL C00479 V=800.0 PL=0
MOVL C00480 V=800.0 PL=0
MOVL C00481 V=800.0 PL=0
MOVL C00482 V=800.0 PL=0
MOVL C00483 V=800.0 PL=0
MOVL C00484 V=800.0 PL=0
MOVL C00485 V=800.0 PL=0
MOVL C00486 V=800.0 PL=0
MOVL C00487 V=800.0 PL=0
MOVL C00488 V=800.0 PL=0
MOVL C00489 V=800.0 PL=0
MOVL C00490 V=800.0 PL=0
MOVL C00491 V=800.0 PL=0
MOVL C00492 V=800.0 PL=0
MOVL C00493 V=800.0 PL=0
MOVL C00494 V=800.0 PL=0
MOVL C00495 V=800.0 PL=0
MOVL C00496 V=800.0 PL=0
MOVL C00497 V=800.0 PL=0
MOVL C00498 V=800.0 PL=0
MOVL C00499 V=800.0 PL=0
MOVL C00500 V=800.0 PL=0
MOVL C00501 V=800.0 PL=0
MOVL C00502 V=800.0 PL=0
MOVL C00503 V=800.0 PL=0
MOVL C00504 V=800.0 PL=0
MOVL C00505 V=800.0 PL=0
MOVL C00506 V=800.0 PL=0
MOVL C00507 V=800.0 PL=0
MOVL C00508 V=800.0 PL=0
MOVL C00509 V=800.0 PL=0
MOVL C00510 V=800.0 PL=0
MOVL C00511 V=800.0 PL=0
MOVL C00512 V=800.0 PL=0
MOVL C00513 V=800.0 PL=0
MOVL C00514 V=800.0 PL=0
MOVL C00515 V=800.0 PL=0
MOVL C00516 V=800.0 PL=0
MOVL C00517 V=800.0 PL=0
MOVL C00518 V=800.0 PL=0
MOVL C00519 V=800.0 PL=0
MOVL C00520 V=800.0 PL=0
MOVL C00521 V=800.0 PL=0
MOVL C00522 V=800.0 PL=0
MOVL C00523 V=800.0 PL=0
MOVL C00524 V=800.0 PL=0
MOVL C00525 V=800.0 PL=0
MOVL C00526 V=800.0 PL=0
MOVL C00527 V=800.0 PL=0
MOVL C00528 V=800.0 PL=0
MOVL C00529 V=800.0 PL=0
MOVL C00530 V=800.0 PL=0
MOVL C00531 V=800.0 PL=0
MOVL C00532 V=800.0 PL=0
MOVL C00533 V=800.0 PL=0
MOVL C00534 V=800.0 PL=0
MOVL C00535 V=800.0 PL=0
MOVL C00536 V=800.0 PL=0
MOVL C00537 V=800.0 PL=0
MOVL C00538 V=800.0 PL=0
MOVL C00539 V=800.0 PL=0
MOVL C00540 V=800.0 PL=0
MOVL C00541 V=800.0 PL=0
MOVL C00542 V=800.0 PL=0
MOVL C00543 V=800.0 PL=0
MOVL C00544 V=800.0 PL=0
MOVL C00545 V=800.0 PL=0
MOVL C00546 V=800.0 PL=0
MOVL C00547 V=800.0 PL=0
MOVL C00548 V=800.0 PL=0
MOVL C00549 V=800.0 PL=0
MOVL C00550 V=800.0 PL=0
MOVL C00551 V=800.0 PL=0
MOVL C00552 V=800.0 PL=0
MOVL C00553 V=800.0 PL=0
MOVL C00554 V=800.0 PL=0
MOVL C00555 V=800.0 PL=0
MOVL C00556 V=800.0 PL=0
MOVL C00557 V=800.0 PL=0
MOVL C00558 V=800.0 PL=0
MOVL C00559 V=800.0 PL=0
MOVL C00560 V=800.0 PL=0
MOVL C00561 V=800.0 PL=0
MOVL C00562 V=800.0 PL=0
MOVL C00563 V=800.0 PL=0
MOVL C00564 V=800.0 PL=0
MOVL C00565 V=800.0 PL=0
MOVL C00566 V=800.0 PL=0
MOVL C00567 V=800.0 PL=0
MOVL C00568 V=800.0 PL=0
MOVL C00569 V=800.0 PL=0
MOVL C00570 V=800.0 PL=0
MOVL C00571 V=800.0 PL=0
MOVL C00572 V=800.0 PL=0
MOVL C00573 V=800.0 PL=0
MOVL C00574 V=800.0 PL=0
MOVL C00575 V=800.0 PL=0
MOVL C00576 V=800.0 PL=0
MOVL C00577 V=800.0 PL=0
MOVL C00578 V=800.0 PL=0
MOVL C00579 V=800.0 PL=0
MOVL C00580 V=800.0 PL=0
MOVL C00581 V=800.0 PL=0
MOVL C00582 V=800.0 PL=0
MOVL C00583 V=800.0 PL=0
MOVL C00584 V=800.0 PL=0
MOVL C00585 V=800.0 PL=0
MOVL C00586 V=800.0 PL=0
MOVL C00587 V=800.0 PL=0
MOVL C00588 V=800.0 PL=0
MOVL C00589 V=800.0 PL=0
MOVL C00590 V=800.0 PL=0
MOVL C00591 V=800.0 PL=0
MOVL C00592 V=800.0 PL=0
MOVL C00593 V=800.0 PL=0
MOVL C00594 V=800.0 PL=0
MOVL C00595 V=800.0 PL=0
MOVL C00596 V=800.0 PL=0
MOVL C00597 V=800.0 PL=0
MOVL C00598 V=800.0 PL=0
MOVL C00599 V=800.0 PL=0
MOVL C00600 V=800.0 PL=0
MOVL C00601 V=800.0 PL=0
MOVL C00602 V=800.0 PL=0
MOVL C00603 V=800.0 PL=0
MOVL C00604 V=800.0 PL=0
MOVL C00605 V=800.0 PL=0
MOVL C00606 V=800.0 PL=0
MOVL C00607 V=800.0 PL=0
MOVL C00608 V=800.0 PL=0
MOVL C00609 V=800.0 PL=0
MOVL C00610 V=800.0 PL=0
MOVL C00611 V=800.0 PL=0
MOVL C00612 V=800.0 PL=0
MOVL C00613 V=800.0 PL=0
MOVL C00614 V=800.0 PL=0
MOVL C00615 V=800.0 PL=0
MOVL C00616 V=800.0 PL=0
MOVL C00617 V=800.0 PL=0
MOVL C00618 V=800.0 PL=0
MOVL C00619 V=800.0 PL=0
MOVL C00620 V=800.0 PL=0
MOVL C00621 V=800.0 PL=0
MOVL C00622 V=800.0 PL=0
MOVL C00623 V=800.0 PL=0
MOVL C00624 V=800.0 PL=0
MOVL C00625 V=800.0 PL=0
MOVL C00626 V=800.0 PL=0
MOVL C00627 V=800.0 PL=0
MOVL C00628 V=800.0 PL=0
MOVL C00629 V=800.0 PL=0
MOVL C00630 V=800.0 PL=0
MOVL C00631 V=800.0 PL=0
MOVL C00632 V=800.0 PL=0
MOVL C00633 V=800.0 PL=0
MOVL C00634 V=800.0 PL=0
MOVL C00635 V=800.0 PL=0
MOVL C00636 V=800.0 PL=0
MOVL C00637 V=800.0 PL=0
MOVL C00638 V=800.0 PL=0
MOVL C00639 V=800.0 PL=0
MOVL C00640 V=800.0 PL=0
MOVL C00641 V=800.0 PL=0
MOVL C00642 V=800.0 PL=0
MOVL C00643 V=800.0 PL=0
MOVL C00644 V=800.0 PL=0
MOVL C00645 V=800.0 PL=0
MOVL C00646 V=800.0 PL=0
MOVL C00647 V=800.0 PL=0
MOVL C00648 V=800.0 PL=0
MOVL C00649 V=800.0 PL=0
MOVL C00650 V=800.0 PL=0
MOVL C00651 V=800.0 PL=0
MOVL C00652 V=800.0 PL=0
MOVL C00653 V=800.0 PL=0
MOVL C00654 V=800.0 PL=0
MOVL C00655 V=800.0 PL=0
MOVL C00656 V=800.0 PL=0
MOVL C00657 V=800.0 PL=0
MOVL C00658 V=800.0 PL=0
MOVL C00659 V=800.0 PL=0
MOVL C00660 V=800.0 PL=0
MOVL C00661 V=800.0 PL=0
MOVL C00662 V=800.0 PL=0
MOVL C00663 V=800.0 PL=0
MOVL C00664 V=800.0 PL=0
MOVL C00665 V=800.0 PL=0
MOVL C00666 V=800.0 PL=0
MOVL C00667 V=800.0 PL=0
MOVL C00668 V=800.0 PL=0
MOVL C00669 V=800.0 PL=0
MOVL C00670 V=800.0 PL=0
MOVL C00671 V=800.0 PL=0
MOVL C00672 V=800.0 PL=0
MOVL C00673 V=800.0 PL=0
MOVL C00674 V=800.0 PL=0
MOVL C00675 V=800.0 PL=0
MOVL C00676 V=800.0 PL=0
MOVL C00677 V=800.0 PL=0
MOVL C00678 V=800.0 PL=0
MOVL C00679 V=800.0 PL=0
MOVL C00680 V=800.0 PL=0
MOVL C00681 V=800.0 PL=0
MOVL C00682 V=800.0 PL=0
MOVL C00683 V=800.0 PL=0
MOVL C00684 V=800.0 PL=0
MOVL C00685 V=800.0 PL=0
MOVL C00686 V=800.0 PL=0
MOVL C00687 V=800.0 PL=0
MOVL C00688 V=800.0 PL=0
MOVL C00689 V=800.0 PL=0
MOVL C00690 V=800.0 PL=0
MOVL C00691 V=800.0 PL=0
MOVL C00692 V=800.0 PL=0
MOVL C00693 V=800.0 PL=0
MOVL C00694 V=800.0 PL=0
MOVL C00695 V=800.0 PL=0
MOVL C00696 V=800.0 PL=0
MOVL C00697 V=800.0 PL=0
MOVL C00698 V=800.0 PL=0
MOVL C00699 V=800.0 PL=0
MOVL C00700 V=800.0 PL=0
MOVL C00701 V=800.0 PL=0
MOVL C00702 V=800.0 PL=0
MOVL C00703 V=800.0 PL=0
MOVL C00704 V=800.0 PL=0
MOVL C00705 V=800.0 PL=0
MOVL C00706 V=800.0 PL=0
MOVL C00707 V=800.0 PL=0
MOVL C00708 V=800.0 PL=0
MOVL C00709 V=800.0 PL=0
MOVL C00710 V=800.0 PL=0
MOVL C00711 V=800.0 PL=0
MOVL C00712 V=800.0 PL=0
MOVL C00713 V=800.0 PL=0
MOVL C00714 V=800.0 PL=0
MOVL C00715 V=800.0 PL=0
MOVL C00716 V=800.0 PL=0
MOVL C00717 V=800.0 PL=0
MOVL C00718 V=800.0 PL=0
MOVL C00719 V=800.0 PL=0
MOVL C00720 V=800.0 PL=0
MOVL C00721 V=800.0 PL=0
MOVL C00722 V=800.0 PL=0
MOVL C00723 V=800.0 PL=0
MOVL C00724 V=800.0 PL=0
MOVL C00725 V=800.0 PL=0
MOVL C00726 V=800.0 PL=0
MOVL C00727 V=800.0 PL=0
MOVL C00728 V=800.0 PL=0
MOVL C00729 V=800.0 PL=0
MOVL C00730 V=800.0 PL=0
MOVL C00731 V=800.0 PL=0
MOVL C00732 V=800.0 PL=0
MOVL C00733 V=800.0 PL=0
MOVL C00734 V=800.0 PL=0
MOVL C00735 V=800.0 PL=0
MOVL C00736 V=800.0 PL=0
MOVL C00737 V=800.0 PL=0
MOVL C00738 V=800.0 PL=0
MOVL C00739 V=800.0 PL=0
MOVL C00740 V=800.0 PL=0
MOVL C00741 V=800.0 PL=0
MOVL C00742 V=800.0 PL=0
MOVL C00743 V=800.0 PL=0
MOVL C00744 V=800.0 PL=0
MOVL C00745 V=800.0 PL=0
MOVL C00746 V=800.0 PL=0
MOVL C00747 V=800.0 PL=0
MOVL C00748 V=800.0 PL=0
MOVL C00749 V=800.0 PL=0
MOVL C00750 V=800.0 PL=0
MOVL C00751 V=800.0 PL=0
MOVL C00752 V=800.0 PL=0
MOVL C00753 V=800.0 PL=0
MOVL C00754 V=800.0 PL=0
MOVL C00755 V=800.0 PL=0
MOVL C00756 V=800.0 PL=0
MOVL C00757 V=800.0 PL=0
MOVL C00758 V=800.0 PL=0
MOVL C00759 V=800.0 PL=0
MOVL C00760 V=800.0 PL=0
MOVL C00761 V=800.0 PL=0
MOVL C00762 V=800.0 PL=0
MOVL C00763 V=800.0 PL=0
MOVL C00764 V=800.0 PL=0
MOVL C00765 V=800.0 PL=0
MOVL C00766 V=800.0 PL=0
MOVL C00767 V=800.0 PL=0
MOVL C00768 V=800.0 PL=0
MOVL C00769 V=800.0 PL=0
MOVL C00770 V=800.0 PL=0
MOVL C00771 V=800.0 PL=0
MOVL C00772 V=800.0 PL=0
MOVL C00773 V=800.0 PL=0
MOVL C00774 V=800.0 PL=0
MOVL C00775 V=800.0 PL=0
MOVL C00776 V=800.0 PL=0
MOVL C00777 V=800.0 PL=0
MOVL C00778 V=800.0 PL=0
MOVL C00779 V=800.0 PL=0
MOVL C00780 V=800.0 PL=0
MOVL C00781 V=800.0 PL=0
MOVL C00782 V=800.0 PL=0
MOVL C00783 V=800.0 PL=0
MOVL C00784 V=800.0 PL=0
MOVL C00785 V=800.0 PL=0
MOVL C00786 V=800.0 PL=0
MOVL C00787 V=800.0 PL=0
MOVL C00788 V=800.0 PL=0
MOVL C00789 V=800.0 PL=0
MOVL C00790 V=800.0 PL=0
MOVL C00791 V=800.0 PL=0
MOVL C00792 V=800.0 PL=0
MOVL C00793 V=800.0 PL=0
MOVL C00794 V=800.0 PL=0
MOVL C00795 V=800.0 PL=0
MOVL C00796 V=800.0 PL=0
MOVL C00797 V=800.0 PL=0
MOVL C00798 V=800.0 PL=0
MOVL C00799 V=800.0 PL=0
MOVL C00800 V=800.0 PL=0
MOVL C00801 V=800.0 PL=0
MOVL C00802 V=800.0 PL=0
MOVL C00803 V=800.0 PL=0
MOVL C00804 V=800.0 PL=0
MOVL C00805 V=800.0 PL=0
MOVL C00806 V=800.0 PL=0
MOVL C00807 V=800.0 PL=0
MOVL C00808 V=800.0 PL=0
MOVL C00809 V=800.0 PL=0
MOVL C00810 V=800.0 PL=0
MOVL C00811 V=800.0 PL=0
MOVL C00812 V=800.0 PL=0
MOVL C00813 V=800.0 PL=0
MOVL C00814 V=800.0 PL=0
MOVL C00815 V=800.0 PL=0
MOVL C00816 V=800.0 PL=0
MOVL C00817 V=800.0 PL=0
MOVL C00818 V=800.0 PL=0
MOVL C00819 V=800.0 PL=0
MOVL C00820 V=800.0 PL=0
MOVL C00821 V=800.0 PL=0
MOVL C00822 V=800.0 PL=0
MOVL C00823 V=800.0 PL=0
MOVL C00824 V=800.0 PL=0
MOVL C00825 V=800.0 PL=0
MOVL C00826 V=800.0 PL=0
MOVL C00827 V=800.0 PL=0
MOVL C00828 V=800.0 PL=0
MOVL C00829 V=800.0 PL=0
MOVL C00830 V=800.0 PL=0
MOVL C00831 V=800.0 PL=0
MOVL C00832 V=800.0 PL=0
MOVL C00833 V=800.0 PL=0
MOVL C00834 V=800.0 PL=0
MOVL C00835 V=800.0 PL=0
MOVL C00836 V=800.0 PL=0
MOVL C00837 V=800.0 PL=0
MOVL C00838 V=800.0 PL=0
MOVL C00839 V=800.0 PL=0
MOVL C00840 V=800.0 PL=0
MOVL C00841 V=800.0 PL=0
MOVL C00842 V=800.0 PL=0
MOVL C00843 V=800.0 PL=0
MOVL C00844 V=800.0 PL=0
MOVL C00845 V=800.0 PL=0
MOVL C00846 V=800.0 PL=0
MOVL C00847 V=800.0 PL=0
MOVL C00848 V=800.0 PL=0
MOVL C00849 V=800.0 PL=0
MOVL C00850 V=800.0 PL=0
MOVL C00851 V=800.0 PL=0
MOVL C00852 V=800.0 PL=0
MOVL C00853 V=800.0 PL=0
MOVL C00854 V=800.0 PL=0
MOVL C00855 V=800.0 PL=0
MOVL C00856 V=800.0 PL=0
MOVL C00857 V=800.0 PL=0
MOVL C00858 V=800.0 PL=0
MOVL C00859 V=800.0 PL=0
MOVL C00860 V=800.0 PL=0
MOVL C00861 V=800.0 PL=0
MOVL C00862 V=800.0 PL=0
MOVL C00863 V=800.0 PL=0
MOVL C00864 V=800.0 PL=0
MOVL C00865 V=800.0 PL=0
MOVL C00866 V=800.0 PL=0
MOVL C00867 V=800.0 PL=0
MOVL C00868 V=800.0 PL=0
MOVL C00869 V=800.0 PL=0
MOVL C00870 V=800.0 PL=0
MOVL C00871 V=800.0 PL=0
MOVL C00872 V=800.0 PL=0
MOVL C00873 V=800.0 PL=0
MOVL C00874 V=800.0 PL=0
MOVL C00875 V=800.0 PL=0
MOVL C00876 V=800.0 PL=0
MOVL C00877 V=800.0 PL=0
MOVL C00878 V=800.0 PL=0
MOVL C00879 V=800.0 PL=0
MOVL C00880 V=800.0 PL=0
MOVL C00881 V=800.0 PL=0
MOVL C00882 V=800.0 PL=0
MOVL C00883 V=800.0 PL=0
MOVL C00884 V=800.0 PL=0
MOVL C00885 V=800.0 PL=0
MOVL C00886 V=800.0 PL=0
MOVL C00887 V=800.0 PL=0
MOVL C00888 V=800.0 PL=0
MOVL C00889 V=800.0 PL=0
MOVL C00890 V=800.0 PL=0
MOVL C00891 V=800.0 PL=0
MOVL C00892 V=800.0 PL=0
MOVL C00893 V=800.0 PL=0
MOVL C00894 V=800.0 PL=0
MOVL C00895 V=800.0 PL=0
MOVL C00896 V=800.0 PL=0
MOVL C00897 V=800.0 PL=0
MOVL C00898 V=800.0 PL=0
MOVL C00899 V=800.0 PL=0
MOVL C00900 V=800.0 PL=0
MOVL C00901 V=800.0 PL=0
MOVL C00902 V=800.0 PL=0
MOVL C00903 V=800.0 PL=0
MOVL C00904 V=800.0 PL=0
MOVL C00905 V=800.0 PL=0
MOVL C00906 V=800.0 PL=0
MOVL C00907 V=800.0 PL=0
MOVL C00908 V=800.0 PL=0
MOVL C00909 V=800.0 PL=0
MOVL C00910 V=800.0 PL=0
MOVL C00911 V=800.0 PL=0
MOVL C00912 V=800.0 PL=0
MOVL C00913 V=800.0 PL=0
MOVL C00914 V=800.0 PL=0
MOVL C00915 V=800.0 PL=0
MOVL C00916 V=800.0 PL=0
MOVL C00917 V=800.0 PL=0
MOVL C00918 V=800.0 PL=0
MOVL C00919 V=800.0 PL=0
MOVL C00920 V=800.0 PL=0
MOVL C00921 V=800.0 PL=0
MOVL C00922 V=800.0 PL=0
MOVL C00923 V=800.0 PL=0
MOVL C00924 V=800.0 PL=0
MOVL C00925 V=800.0 PL=0
MOVL C00926 V=800.0 PL=0
MOVL C00927 V=800.0 PL=0
MOVL C00928 V=800.0 PL=0
MOVL C00929 V=800.0 PL=0
MOVL C00930 V=800.0 PL=0
MOVL C00931 V=800.0 PL=0
MOVL C00932 V=800.0 PL=0
MOVL C00933 V=800.0 PL=0
MOVL C00934 V=800.0 PL=0
MOVL C00935 V=800.0 PL=0
MOVL C00936 V=800.0 PL=0
MOVL C00937 V=800.0 PL=0
MOVL C00938 V=800.0 PL=0
MOVL C00939 V=800.0 PL=0
MOVL C00940 V=800.0 PL=0
MOVL C00941 V=800.0 PL=0
MOVL C00942 V=800.0 PL=0
MOVL C00943 V=800.0 PL=0
MOVL C00944 V=800.0 PL=0
MOVL C00945 V=800.0 PL=0
MOVL C00946 V=800.0 PL=0
MOVL C00947 V=800.0 PL=0
MOVL C00948 V=800.0 PL=0
MOVL C00949 V=800.0 PL=0
MOVL C00950 V=800.0 PL=0
MOVL C00951 V=800.0 PL=0
MOVL C00952 V=800.0 PL=0
MOVL C00953 V=800.0 PL=0
MOVL C00954 V=800.0 PL=0
MOVL C00955 V=800.0 PL=0
MOVL C00956 V=800.0 PL=0
MOVL C00957 V=800.0 PL=0
MOVL C00958 V=800.0 PL=0
MOVL C00959 V=800.0 PL=0
MOVL C00960 V=800.0 PL=0
MOVL C00961 V=800.0 PL=0
MOVL C00962 V=800.0 PL=0
MOVL C00963 V=800.0 PL=0
MOVL C00964 V=800.0 PL=0
MOVL C00965 V=800.0 PL=0
MOVL C00966 V=800.0 PL=0
MOVL C00967 V=800.0 PL=0
MOVL C00968 V=800.0 PL=0
MOVL C00969 V=800.0 PL=0
MOVL C00970 V=800.0 PL=0
MOVL C00971 V=800.0 PL=0
MOVL C00972 V=800.0 PL=0
MOVL C00973 V=800.0 PL=0
MOVL C00974 V=800.0 PL=0
MOVL C00975 V=800.0 PL=0
MOVL C00976 V=800.0 PL=0
MOVL C00977 V=800.0 PL=0
MOVL C00978 V=800.0 PL=0
MOVL C00979 V=800.0 PL=0
MOVL C00980 V=800.0 PL=0
MOVL C00981 V=800.0 PL=0
MOVL C00982 V=800.0 PL=0
MOVL C00983 V=800.0 PL=0
MOVL C00984 V=800.0 PL=0
MOVL C00985 V=800.0 PL=0
MOVL C00986 V=800.0 PL=0
MOVL C00987 V=800.0 PL=0
MOVL C00988 V=800.0 PL=0
MOVL C00989 V=800.0 PL=0
MOVL C00990 V=800.0 PL=0
MOVL C00991 V=800.0 PL=0
MOVL C00992 V=800.0 PL=0
MOVL C00993 V=800.0 PL=0
MOVL C00994 V=800.0 PL=0
MOVL C00995 V=800.0 PL=0
MOVL C00996 V=800.0 PL=0
MOVL C00997 V=800.0 PL=0
MOVL C00998 V=800.0 PL=0
MOVL C00999 V=800.0 PL=0
MOVL C01000 V=800.0 PL=0
MOVL C01001 V=800.0 PL=0
MOVL C01002 V=800.0 PL=0
MOVL C01003 V=800.0 PL=0
MOVL C01004 V=800.0 PL=0
MOVL C01005 V=800.0 PL=0
MOVL C01006 V=800.0 PL=0
MOVL C01007 V=800.0 PL=0
MOVL C01008 V=800.0 PL=0
MOVL C01009 V=800.0 PL=0
MOVL C01010 V=800.0 PL=0
MOVL C01011 V=800.0 PL=0
MOVL C01012 V=800.0 PL=0
MOVL C01013 V=800.0 PL=0
MOVL C01014 V=800.0 PL=0
MOVL C01015 V=800.0 PL=0
MOVL C01016 V=800.0 PL=0
MOVL C01017 V=800.0 PL=0
MOVL C01018 V=800.0 PL=0
MOVL C01019 V=800.0 PL=0
MOVL C01020 V=800.0 PL=0
MOVL C01021 V=800.0 PL=0
MOVL C01022 V=800.0 PL=0
MOVL C01023 V=800.0 PL=0
MOVL C01024 V=800.0 PL=0
MOVL C01025 V=800.0 PL=0
MOVL C01026 V=800.0 PL=0
MOVL C01027 V=800.0 PL=0
MOVL C01028 V=800.0 PL=0
MOVL C01029 V=800.0 PL=0
MOVL C01030 V=800.0 PL=0
MOVL C01031 V=800.0 PL=0
MOVL C01032 V=800.0 PL=0
MOVL C01033 V=800.0 PL=0
MOVL C01034 V=800.0 PL=0
MOVL C01035 V=800.0 PL=0
MOVL C01036 V=800.0 PL=0
MOVL C01037 V=800.0 PL=0
MOVL C01038 V=800.0 PL=0
MOVL C01039 V=800.0 PL=0
MOVL C01040 V=800.0 PL=0
MOVL C01041 V=800.0 PL=0
MOVL C01042 V=800.0 PL=0
MOVL C01043 V=800.0 PL=0
MOVL C01044 V=800.0 PL=0
MOVL C01045 V=800.0 PL=0
MOVL C01046 V=800.0 PL=0
MOVL C01047 V=800.0 PL=0
MOVL C01048 V=800.0 PL=0
MOVL C01049 V=800.0 PL=0
MOVL C01050 V=800.0 PL=0
MOVL C01051 V=800.0 PL=0
MOVL C01052 V=800.0 PL=0
MOVL C01053 V=800.0 PL=0
MOVL C01054 V=800.0 PL=0
MOVL C01055 V=800.0 PL=0
MOVL C01056 V=800.0 PL=0
MOVL C01057 V=800.0 PL=0
MOVL C01058 V=800.0 PL=0
MOVL C01059 V=800.0 PL=0
MOVL C01060 V=800.0 PL=0
MOVL C01061 V=800.0 PL=0
MOVL C01062 V=800.0 PL=0
MOVL C01063 V=800.0 PL=0
MOVL C01064 V=800.0 PL=0
MOVL C01065 V=800.0 PL=0
MOVL C01066 V=800.0 PL=0
MOVL C01067 V=800.0 PL=0
MOVL C01068 V=800.0 PL=0
MOVL C01069 V=800.0 PL=0
MOVL C01070 V=800.0 PL=0
MOVL C01071 V=800.0 PL=0
MOVL C01072 V=800.0 PL=0
MOVL C01073 V=800.0 PL=0
MOVL C01074 V=800.0 PL=0
MOVL C01075 V=800.0 PL=0
MOVL C01076 V=800.0 PL=0
MOVL C01077 V=800.0 PL=0
MOVL C01078 V=800.0 PL=0
MOVL C01079 V=800.0 PL=0
MOVL C01080 V=800.0 PL=0
MOVL C01081 V=800.0 PL=0
MOVL C01082 V=800.0 PL=0
MOVL C01083 V=800.0 PL=0
MOVL C01084 V=800.0 PL=0
MOVL C01085 V=800.0 PL=0
MOVL C01086 V=800.0 PL=0
MOVL C01087 V=800.0 PL=0
MOVL C01088 V=800.0 PL=0
MOVL C01089 V=800.0 PL=0
MOVL C01090 V=800.0 PL=0
MOVL C01091 V=800.0 PL=0
MOVL C01092 V=800.0 PL=0
MOVL C01093 V=800.0 PL=0
MOVL C01094 V=800.0 PL=0
MOVL C01095 V=800.0 PL=0
MOVL C01096 V=800.0 PL=0
MOVL C01097 V=800.0 PL=0
MOVL C01098 V=800.0 PL=0
MOVL C01099 V=800.0 PL=0
MOVL C01100 V=800.0 PL=0
MOVL C01101 V=800.0 PL=0
MOVL C01102 V=800.0 PL=0
MOVL C01103 V=800.0 PL=0
MOVL C01104 V=800.0 PL=0
MOVL C01105 V=800.0 PL=0
MOVL C01106 V=800.0 PL=0
MOVL C01107 V=800.0 PL=0
MOVL C01108 V=800.0 PL=0
MOVL C01109 V=800.0 PL=0
MOVL C01110 V=800.0 PL=0
MOVL C01111 V=800.0 PL=0
MOVL C01112 V=800.0 PL=0
MOVL C01113 V=800.0 PL=0
MOVL C01114 V=800.0 PL=0
MOVL C01115 V=800.0 PL=0
MOVL C01116 V=800.0 PL=0
MOVL C01117 V=800.0 PL=0
MOVL C01118 V=800.0 PL=0
MOVL C01119 V=800.0 PL=0
MOVL C01120 V=800.0 PL=0
MOVL C01121 V=800.0 PL=0
MOVL C01122 V=800.0 PL=0
MOVL C01123 V=800.0 PL=0
MOVL C01124 V=800.0 PL=0
MOVL C01125 V=800.0 PL=0
MOVL C01126 V=800.0 PL=0
MOVL C01127 V=800.0 PL=0
MOVL C01128 V=800.0 PL=0
MOVL C01129 V=800.0 PL=0
MOVL C01130 V=800.0 PL=0
MOVL C01131 V=800.0 PL=0
MOVL C01132 V=800.0 PL=0
MOVL C01133 V=800.0 PL=0
MOVL C01134 V=800.0 PL=0
MOVL C01135 V=800.0 PL=0
MOVL C01136 V=800.0 PL=0
MOVL C01137 V=800.0 PL=0
MOVL C01138 V=800.0 PL=0
MOVL C01139 V=800.0 PL=0
MOVL C01140 V=800.0 PL=0
MOVL C01141 V=800.0 PL=0
MOVL C01142 V=800.0 PL=0
MOVL C01143 V=800.0 PL=0
MOVL C01144 V=800.0 PL=0
MOVL C01145 V=800.0 PL=0
MOVL C01146 V=800.0 PL=0
MOVL C01147 V=800.0 PL=0
MOVL C01148 V=800.0 PL=0
MOVL C01149 V=800.0 PL=0
MOVL C01150 V=800.0 PL=0
MOVL C01151 V=800.0 PL=0
MOVL C01152 V=800.0 PL=0
MOVL C01153 V=800.0 PL=0
MOVL C01154 V=800.0 PL=0
MOVL C01155 V=800.0 PL=0
MOVL C01156 V=800.0 PL=0
MOVL C01157 V=800.0 PL=0
MOVL C01158 V=800.0 PL=0
MOVL C01159 V=800.0 PL=0
MOVL C01160 V=800.0 PL=0
MOVL C01161 V=800.0 PL=0
MOVL C01162 V=800.0 PL=0
MOVL C01163 V=800.0 PL=0
MOVL C01164 V=800.0 PL=0
MOVL C01165 V=800.0 PL=0
MOVL C01166 V=800.0 PL=0
MOVL C01167 V=800.0 PL=0
MOVL C01168 V=800.0 PL=0
MOVL C01169 V=800.0 PL=0
MOVL C01170 V=800.0 PL=0
MOVL C01171 V=800.0 PL=0
MOVL C01172 V=800.0 PL=0
MOVL C01173 V=800.0 PL=0
MOVL C01174 V=800.0 PL=0
MOVL C01175 V=800.0 PL=0
MOVL C01176 V=800.0 PL=0
MOVL C01177 V=800.0 PL=0
MOVL C01178 V=800.0 PL=0
MOVL C01179 V=800.0 PL=0
MOVL C01180 V=800.0 PL=0
MOVL C01181 V=800.0 PL=0
MOVL C01182 V=800.0 PL=0
MOVL C01183 V=800.0 PL=0
MOVL C01184 V=800.0 PL=0
MOVL C01185 V=800.0 PL=0
MOVL C01186 V=800.0 PL=0
MOVL C01187 V=800.0 PL=0
MOVL C01188 V=800.0 PL=0
MOVL C01189 V=800.0 PL=0
MOVL C01190 V=800.0 PL=0
MOVL C01191 V=800.0 PL=0
MOVL C01192 V=800.0 PL=0
MOVL C01193 V=800.0 PL=0
MOVL C01194 V=800.0 PL=0
MOVL C01195 V=800.0 PL=0
MOVL C01196 V=800.0 PL=0
MOVL C01197 V=800.0 PL=0
MOVL C01198 V=800.0 PL=0
MOVL C01199 V=800.0 PL=0
MOVL C01200 V=800.0 PL=0
MOVL C01201 V=800.0 PL=0
MOVL C01202 V=800.0 PL=0
MOVL C01203 V=800.0 PL=0
MOVL C01204 V=800.0 PL=0
MOVL C01205 V=800.0 PL=0
MOVL C01206 V=800.0 PL=0
MOVL C01207 V=800.0 PL=0
MOVL C01208 V=800.0 PL=0
MOVL C01209 V=800.0 PL=0
MOVL C01210 V=800.0 PL=0
MOVL C01211 V=800.0 PL=0
MOVL C01212 V=800.0 PL=0
MOVL C01213 V=800.0 PL=0
MOVL C01214 V=800.0 PL=0
MOVL C01215 V=800.0 PL=0
MOVL C01216 V=800.0 PL=0
MOVL C01217 V=800.0 PL=0
MOVL C01218 V=800.0 PL=0
MOVL C01219 V=800.0 PL=0
MOVL C01220 V=800.0 PL=0
MOVL C01221 V=800.0 PL=0
MOVL C01222 V=800.0 PL=0
MOVL C01223 V=800.0 PL=0
MOVL C01224 V=800.0 PL=0
MOVL C01225 V=800.0 PL=0
MOVL C01226 V=800.0 PL=0
MOVL C01227 V=800.0 PL=0
MOVL C01228 V=800.0 PL=0
MOVL C01229 V=800.0 PL=0
MOVL C01230 V=800.0 PL=0
MOVL C01231 V=800.0 PL=0
MOVL C01232 V=800.0 PL=0
MOVL C01233 V=800.0 PL=0
MOVL C01234 V=800.0 PL=0
MOVL C01235 V=800.0 PL=0
MOVL C01236 V=800.0 PL=0
MOVL C01237 V=800.0 PL=0
MOVL C01238 V=800.0 PL=0
MOVL C01239 V=800.0 PL=0
MOVL C01240 V=800.0 PL=0
MOVL C01241 V=800.0 PL=0
MOVL C01242 V=800.0 PL=0
MOVL C01243 V=800.0 PL=0
MOVL C01244 V=800.0 PL=0
MOVL C01245 V=800.0 PL=0
MOVL C01246 V=800.0 PL=0
MOVL C01247 V=800.0 PL=0
MOVL C01248 V=800.0 PL=0
MOVL C01249 V=800.0 PL=0
MOVL C01250 V=800.0 PL=0
MOVL C01251 V=800.0 PL=0
MOVL C01252 V=800.0 PL=0
MOVL C01253 V=800.0 PL=0
MOVL C01254 V=800.0 PL=0
MOVL C01255 V=800.0 PL=0
MOVL C01256 V=800.0 PL=0
MOVL C01257 V=800.0 PL=0
MOVL C01258 V=800.0 PL=0
MOVL C01259 V=800.0 PL=0
MOVL C01260 V=800.0 PL=0
MOVL C01261 V=800.0 PL=0
MOVL C01262 V=800.0 PL=0
MOVL C01263 V=800.0 PL=0
MOVL C01264 V=800.0 PL=0
MOVL C01265 V=800.0 PL=0
MOVL C01266 V=800.0 PL=0
MOVL C01267 V=800.0 PL=0
MOVL C01268 V=800.0 PL=0
MOVL C01269 V=800.0 PL=0
MOVL C01270 V=800.0 PL=0
MOVL C01271 V=800.0 PL=0
MOVL C01272 V=800.0 PL=0
MOVL C01273 V=800.0 PL=0
MOVL C01274 V=800.0 PL=0
MOVL C01275 V=800.0 PL=0
MOVL C01276 V=800.0 PL=0
MOVL C01277 V=800.0 PL=0
MOVL C01278 V=800.0 PL=0
MOVL C01279 V=800.0 PL=0
MOVL C01280 V=800.0 PL=0
MOVL C01281 V=800.0 PL=0
MOVL C01282 V=800.0 PL=0
MOVL C01283 V=800.0 PL=0
MOVL C01284 V=800.0 PL=0
MOVL C01285 V=800.0 PL=0
MOVL C01286 V=800.0 PL=0
MOVL C01287 V=800.0 PL=0
MOVL C01288 V=800.0 PL=0
MOVL C01289 V=800.0 PL=0
MOVL C01290 V=800.0 PL=0
MOVL C01291 V=800.0 PL=0
MOVL C01292 V=800.0 PL=0
MOVL C01293 V=800.0 PL=0
MOVL C01294 V=800.0 PL=0
MOVL C01295 V=800.0 PL=0
MOVL C01296 V=800.0 PL=0
MOVL C01297 V=800.0 PL=0
MOVL C01298 V=800.0 PL=0
MOVL C01299 V=800.0 PL=0
MOVL C01300 V=800.0 PL=0
MOVL C01301 V=800.0 PL=0
MOVL C01302 V=800.0 PL=0
MOVL C01303 V=800.0 PL=0
MOVL C01304 V=800.0 PL=0
MOVL C01305 V=800.0 PL=0
MOVL C01306 V=800.0 PL=0
MOVL C01307 V=800.0 PL=0
MOVL C01308 V=800.0 PL=0
MOVL C01309 V=800.0 PL=0
MOVL C01310 V=800.0 PL=0
MOVL C01311 V=800.0 PL=0
MOVL C01312 V=800.0 PL=0
MOVL C01313 V=800.0 PL=0
MOVL C01314 V=800.0 PL=0
MOVL C01315 V=800.0 PL=0
MOVL C01316 V=800.0 PL=0
MOVL C01317 V=800.0 PL=0
MOVL C01318 V=800.0 PL=0
MOVL C01319 V=800.0 PL=0
MOVL C01320 V=800.0 PL=0
MOVL C01321 V=800.0 PL=0
MOVL C01322 V=800.0 PL=0
MOVL C01323 V=800.0 PL=0
MOVL C01324 V=800.0 PL=0
MOVL C01325 V=800.0 PL=0
MOVL C01326 V=800.0 PL=0
MOVL C01327 V=800.0 PL=0
MOVL C01328 V=800.0 PL=0
MOVL C01329 V=800.0 PL=0
MOVL C01330 V=800.0 PL=0
MOVL C01331 V=800.0 PL=0
MOVL C01332 V=800.0 PL=0
MOVL C01333 V=800.0 PL=0
MOVL C01334 V=800.0 PL=0
MOVL C01335 V=800.0 PL=0
MOVL C01336 V=800.0 PL=0
MOVL C01337 V=800.0 PL=0
MOVL C01338 V=800.0 PL=0
MOVL C01339 V=800.0 PL=0
MOVL C01340 V=800.0 PL=0
MOVL C01341 V=800.0 PL=0
MOVL C01342 V=800.0 PL=0
MOVL C01343 V=800.0 PL=0
MOVL C01344 V=800.0 PL=0
MOVL C01345 V=800.0 PL=0
MOVL C01346 V=800.0 PL=0
MOVL C01347 V=800.0 PL=0
MOVL C01348 V=800.0 PL=0
MOVL C01349 V=800.0 PL=0
MOVL C01350 V=800.0 PL=0
MOVL C01351 V=800.0 PL=0
MOVL C01352 V=800.0 PL=0
MOVL C01353 V=800.0 PL=0
MOVL C01354 V=800.0 PL=0
MOVL C01355 V=800.0 PL=0
MOVL C01356 V=800.0 PL=0
MOVL C01357 V=800.0 PL=0
MOVL C01358 V=800.0 PL=0
MOVL C01359 V=800.0 PL=0
MOVL C01360 V=800.0 PL=0
MOVL C01361 V=800.0 PL=0
MOVL C01362 V=800.0 PL=0
MOVL C01363 V=800.0 PL=0
MOVL C01364 V=800.0 PL=0
MOVL C01365 V=800.0 PL=0
MOVL C01366 V=800.0 PL=0
MOVL C01367 V=800.0 PL=0
MOVL C01368 V=800.0 PL=0
MOVL C01369 V=800.0 PL=0
MOVL C01370 V=800.0 PL=0
MOVL C01371 V=800.0 PL=0
MOVL C01372 V=800.0 PL=0
MOVL C01373 V=800.0 PL=0
MOVL C01374 V=800.0 PL=0
MOVL C01375 V=800.0 PL=0
MOVL C01376 V=800.0 PL=0
MOVL C01377 V=800.0 PL=0
MOVL C01378 V=800.0 PL=0
MOVL C01379 V=800.0 PL=0
MOVL C01380 V=800.0 PL=0
MOVL C01381 V=800.0 PL=0
MOVL C01382 V=800.0 PL=0
MOVL C01383 V=800.0 PL=0
MOVL C01384 V=800.0 PL=0
MOVL C01385 V=800.0 PL=0
MOVL C01386 V=800.0 PL=0
MOVL C01387 V=800.0 PL=0
MOVL C01388 V=800.0 PL=0
MOVL C01389 V=800.0 PL=0
MOVL C01390 V=800.0 PL=0
MOVL C01391 V=800.0 PL=0
MOVL C01392 V=800.0 PL=0
MOVL C01393 V=800.0 PL=0
MOVL C01394 V=800.0 PL=0
MOVL C01395 V=800.0 PL=0
MOVL C01396 V=800.0 PL=0
MOVL C01397 V=800.0 PL=0
MOVL C01398 V=800.0 PL=0
MOVL C01399 V=800.0 PL=0
MOVL C01400 V=800.0 PL=0
MOVL C01401 V=800.0 PL=0
MOVL C01402 V=800.0 PL=0
MOVL C01403 V=800.0 PL=0
MOVL C01404 V=800.0 PL=0
MOVL C01405 V=800.0 PL=0
MOVL C01406 V=800.0 PL=0
MOVL C01407 V=800.0 PL=0
MOVL C01408 V=800.0 PL=0
MOVL C01409 V=800.0 PL=0
MOVL C01410 V=800.0 PL=0
MOVL C01411 V=800.0 PL=0
MOVL C01412 V=800.0 PL=0
MOVL C01413 V=800.0 PL=0
MOVL C01414 V=800.0 PL=0
MOVL C01415 V=800.0 PL=0
MOVL C01416 V=800.0 PL=0
MOVL C01417 V=800.0 PL=0
MOVL C01418 V=800.0 PL=0
MOVL C01419 V=800.0 PL=0
MOVL C01420 V=800.0 PL=0
MOVL C01421 V=800.0 PL=0
MOVL C01422 V=800.0 PL=0
MOVL C01423 V=800.0 PL=0
MOVL C01424 V=800.0 PL=0
MOVL C01425 V=800.0 PL=0
MOVL C01426 V=800.0 PL=0
MOVL C01427 V=800.0 PL=0
MOVL C01428 V=800.0 PL=0
MOVL C01429 V=800.0 PL=0
MOVL C01430 V=800.0 PL=0
MOVL C01431 V=800.0 PL=0
MOVL C01432 V=800.0 PL=0
MOVL C01433 V=800.0 PL=0
MOVL C01434 V=800.0 PL=0
MOVL C01435 V=800.0 PL=0
MOVL C01436 V=800.0 PL=0
MOVL C01437 V=800.0 PL=0
MOVL C01438 V=800.0 PL=0
MOVL C01439 V=800.0 PL=0
MOVL C01440 V=800.0 PL=0
MOVL C01441 V=800.0 PL=0
MOVL C01442 V=800.0 PL=0
MOVL C01443 V=800.0 PL=0
MOVL C01444 V=800.0 PL=0
MOVL C01445 V=800.0 PL=0
MOVL C01446 V=800.0 PL=0
MOVL C01447 V=800.0 PL=0
MOVL C01448 V=800.0 PL=0
MOVL C01449 V=800.0 PL=0
MOVL C01450 V=800.0 PL=0
MOVL C01451 V=800.0 PL=0
MOVL C01452 V=800.0 PL=0
MOVL C01453 V=800.0 PL=0
MOVL C01454 V=800.0 PL=0
MOVL C01455 V=800.0 PL=0
MOVL C01456 V=800.0 PL=0
MOVL C01457 V=800.0 PL=0
MOVL C01458 V=800.0 PL=0
MOVL C01459 V=800.0 PL=0
MOVL C01460 V=800.0 PL=0
MOVL C01461 V=800.0 PL=0
MOVL C01462 V=800.0 PL=0
MOVL C01463 V=800.0 PL=0
MOVL C01464 V=800.0 PL=0
MOVL C01465 V=800.0 PL=0
MOVL C01466 V=800.0 PL=0
MOVL C01467 V=800.0 PL=0
MOVL C01468 V=800.0 PL=0
MOVL C01469 V=800.0 PL=0
MOVL C01470 V=800.0 PL=0
MOVL C01471 V=800.0 PL=0
MOVL C01472 V=800.0 PL=0
MOVL C01473 V=800.0 PL=0
MOVL C01474 V=800.0 PL=0
MOVL C01475 V=800.0 PL=0
MOVL C01476 V=800.0 PL=0
MOVL C01477 V=800.0 PL=0
MOVL C01478 V=800.0 PL=0
MOVL C01479 V=800.0 PL=0
MOVL C01480 V=800.0 PL=0
MOVL C01481 V=800.0 PL=0
MOVL C01482 V=800.0 PL=0
MOVL C01483 V=800.0 PL=0
MOVL C01484 V=800.0 PL=0
MOVL C01485 V=800.0 PL=0
MOVL C01486 V=800.0 PL=0
MOVL C01487 V=800.0 PL=0
MOVL C01488 V=800.0 PL=0
MOVL C01489 V=800.0 PL=0
MOVL C01490 V=800.0 PL=0
MOVL C01491 V=800.0 PL=0
MOVL C01492 V=800.0 PL=0
MOVL C01493 V=800.0 PL=0
MOVL C01494 V=800.0 PL=0
MOVL C01495 V=800.0 PL=0
MOVL C01496 V=800.0 PL=0
MOVL C01497 V=800.0 PL=0
MOVL C01498 V=800.0 PL=0
MOVL C01499 V=800.0 PL=0
MOVL C01500 V=800.0 PL=0
MOVL C01501 V=800.0 PL=0
MOVL C01502 V=800.0 PL=0
MOVL C01503 V=800.0 PL=0
MOVL C01504 V=800.0 PL=0
MOVL C01505 V=800.0 PL=0
MOVL C01506 V=800.0 PL=0
MOVL C01507 V=800.0 PL=0
MOVL C01508 V=800.0 PL=0
MOVL C01509 V=800.0 PL=0
MOVL C01510 V=800.0 PL=0
MOVL C01511 V=800.0 PL=0
MOVL C01512 V=800.0 PL=0
MOVL C01513 V=800.0 PL=0
MOVL C01514 V=800.0 PL=0
MOVL C01515 V=800.0 PL=0
MOVL C01516 V=800.0 PL=0
MOVL C01517 V=800.0 PL=0
MOVL C01518 V=800.0 PL=0
MOVL C01519 V=800.0 PL=0
MOVL C01520 V=800.0 PL=0
MOVL C01521 V=800.0 PL=0
MOVL C01522 V=800.0 PL=0
MOVL C01523 V=800.0 PL=0
MOVL C01524 V=800.0 PL=0
MOVL C01525 V=800.0 PL=0
MOVL C01526 V=800.0 PL=0
MOVL C01527 V=800.0 PL=0
MOVL C01528 V=800.0 PL=0
MOVL C01529 V=800.0 PL=0
MOVL C01530 V=800.0 PL=0
MOVL C01531 V=800.0 PL=0
MOVL C01532 V=800.0 PL=0
MOVL C01533 V=800.0 PL=0
MOVL C01534 V=800.0 PL=0
MOVL C01535 V=800.0 PL=0
MOVL C01536 V=800.0 PL=0
MOVL C01537 V=800.0 PL=0
MOVL C01538 V=800.0 PL=0
MOVL C01539 V=800.0 PL=0
MOVL C01540 V=800.0 PL=0
MOVL C01541 V=800.0 PL=0
MOVL C01542 V=800.0 PL=0
MOVL C01543 V=800.0 PL=0
MOVL C01544 V=800.0 PL=0
MOVL C01545 V=800.0 PL=0
MOVL C01546 V=800.0 PL=0
MOVL C01547 V=800.0 PL=0
MOVL C01548 V=800.0 PL=0
MOVL C01549 V=800.0 PL=0
MOVL C01550 V=800.0 PL=0
MOVL C01551 V=800.0 PL=0
MOVL C01552 V=800.0 PL=0
MOVL C01553 V=800.0 PL=0
MOVL C01554 V=800.0 PL=0
MOVL C01555 V=800.0 PL=0
MOVL C01556 V=800.0 PL=0
MOVL C01557 V=800.0 PL=0
MOVL C01558 V=800.0 PL=0
MOVL C01559 V=800.0 PL=0
MOVL C01560 V=800.0 PL=0
MOVL C01561 V=800.0 PL=0
MOVL C01562 V=800.0 PL=0
MOVL C01563 V=800.0 PL=0
MOVL C01564 V=800.0 PL=0
MOVL C01565 V=800.0 PL=0
MOVL C01566 V=800.0 PL=0
MOVL C01567 V=800.0 PL=0
MOVL C01568 V=800.0 PL=0
MOVL C01569 V=800.0 PL=0
MOVL C01570 V=800.0 PL=0
MOVL C01571 V=800.0 PL=0
MOVL C01572 V=800.0 PL=0
MOVL C01573 V=800.0 PL=0
MOVL C01574 V=800.0 PL=0
MOVL C01575 V=800.0 PL=0
MOVL C01576 V=800.0 PL=0
MOVL C01577 V=800.0 PL=0
MOVL C01578 V=800.0 PL=0
MOVL C01579 V=800.0 PL=0
MOVL C01580 V=800.0 PL=0
MOVL C01581 V=800.0 PL=0
MOVL C01582 V=800.0 PL=0
MOVL C01583 V=800.0 PL=0
MOVL C01584 V=800.0 PL=0
MOVL C01585 V=800.0 PL=0
MOVL C01586 V=800.0 PL=0
MOVL C01587 V=800.0 PL=0
MOVL C01588 V=800.0 PL=0
MOVL C01589 V=800.0 PL=0
MOVL C01590 V=800.0 PL=0
MOVL C01591 V=800.0 PL=0
MOVL C01592 V=800.0 PL=0
MOVL C01593 V=800.0 PL=0
MOVL C01594 V=800.0 PL=0
MOVL C01595 V=800.0 PL=0
MOVL C01596 V=800.0 PL=0
MOVL C01597 V=800.0 PL=0
MOVL C01598 V=800.0 PL=0
MOVL C01599 V=800.0 PL=0
MOVL C01600 V=800.0 PL=0
MOVL C01601 V=800.0 PL=0
MOVL C01602 V=800.0 PL=0
MOVL C01603 V=800.0 PL=0
MOVL C01604 V=800.0 PL=0
MOVL C01605 V=800.0 PL=0
MOVL C01606 V=800.0 PL=0
MOVL C01607 V=800.0 PL=0
MOVL C01608 V=800.0 PL=0
MOVL C01609 V=800.0 PL=0
MOVL C01610 V=800.0 PL=0
MOVL C01611 V=800.0 PL=0
MOVL C01612 V=800.0 PL=0
MOVL C01613 V=800.0 PL=0
MOVL C01614 V=800.0 PL=0
MOVL C01615 V=800.0 PL=0
MOVL C01616 V=800.0 PL=0
MOVL C01617 V=800.0 PL=0
MOVL C01618 V=800.0 PL=0
MOVL C01619 V=800.0 PL=0
MOVL C01620 V=800.0 PL=0
MOVL C01621 V=800.0 PL=0
MOVL C01622 V=800.0 PL=0
MOVL C01623 V=800.0 PL=0
MOVL C01624 V=800.0 PL=0
MOVL C01625 V=800.0 PL=0
MOVL C01626 V=800.0 PL=0
MOVL C01627 V=800.0 PL=0
MOVL C01628 V=800.0 PL=0
MOVL C01629 V=800.0 PL=0
MOVL C01630 V=800.0 PL=0
MOVL C01631 V=800.0 PL=0
MOVL C01632 V=800.0 PL=0
MOVL C01633 V=800.0 PL=0
MOVL C01634 V=800.0 PL=0
MOVL C01635 V=800.0 PL=0
MOVL C01636 V=800.0 PL=0
MOVL C01637 V=800.0 PL=0
MOVL C01638 V=800.0 PL=0
MOVL C01639 V=800.0 PL=0
MOVL C01640 V=800.0 PL=0
MOVL C01641 V=800.0 PL=0
MOVL C01642 V=800.0 PL=0
MOVL C01643 V=800.0 PL=0
MOVL C01644 V=800.0 PL=0
MOVL C01645 V=800.0 PL=0
MOVL C01646 V=800.0 PL=0
MOVL C01647 V=800.0 PL=0
MOVL C01648 V=800.0 PL=0
MOVL C01649 V=800.0 PL=0
MOVL C01650 V=800.0 PL=0
MOVL C01651 V=800.0 PL=0
MOVL C01652 V=800.0 PL=0
MOVL C01653 V=800.0 PL=0
MOVL C01654 V=800.0 PL=0
MOVL C01655 V=800.0 PL=0
MOVL C01656 V=800.0 PL=0
MOVL C01657 V=800.0 PL=0
MOVL C01658 V=800.0 PL=0
MOVL C01659 V=800.0 PL=0
MOVL C01660 V=800.0 PL=0
MOVL C01661 V=800.0 PL=0
MOVL C01662 V=800.0 PL=0
MOVL C01663 V=800.0 PL=0
MOVL C01664 V=800.0 PL=0
MOVL C01665 V=800.0 PL=0
MOVL C01666 V=800.0 PL=0
MOVL C01667 V=800.0 PL=0
MOVL C01668 V=800.0 PL=0
MOVL C01669 V=800.0 PL=0
MOVL C01670 V=800.0 PL=0
MOVL C01671 V=800.0 PL=0
MOVL C01672 V=800.0 PL=0
MOVL C01673 V=800.0 PL=0
MOVL C01674 V=800.0 PL=0
MOVL C01675 V=800.0 PL=0
MOVL C01676 V=800.0 PL=0
MOVL C01677 V=800.0 PL=0
MOVL C01678 V=800.0 PL=0
MOVL C01679 V=800.0 PL=0
MOVL C01680 V=800.0 PL=0
MOVL C01681 V=800.0 PL=0
MOVL C01682 V=800.0 PL=0
MOVL C01683 V=800.0 PL=0
MOVL C01684 V=800.0 PL=0
MOVL C01685 V=800.0 PL=0
MOVL C01686 V=800.0 PL=0
MOVL C01687 V=800.0 PL=0
MOVL C01688 V=800.0 PL=0
MOVL C01689 V=800.0 PL=0
MOVL C01690 V=800.0 PL=0
MOVL C01691 V=800.0 PL=0
MOVL C01692 V=800.0 PL=0
MOVL C01693 V=800.0 PL=0
MOVL C01694 V=800.0 PL=0
MOVL C01695 V=800.0 PL=0
MOVL C01696 V=800.0 PL=0
MOVL C01697 V=800.0 PL=0
MOVL C01698 V=800.0 PL=0
MOVL C01699 V=800.0 PL=0
MOVL C01700 V=800.0 PL=0
MOVL C01701 V=800.0 PL=0
MOVL C01702 V=800.0 PL=0
MOVL C01703 V=800.0 PL=0
MOVL C01704 V=800.0 PL=0
MOVL C01705 V=800.0 PL=0
MOVL C01706 V=800.0 PL=0
MOVL C01707 V=800.0 PL=0
MOVL C01708 V=800.0 PL=0
MOVL C01709 V=800.0 PL=0
MOVL C01710 V=800.0 PL=0
MOVL C01711 V=800.0 PL=0
MOVL C01712 V=800.0 PL=0
MOVL C01713 V=800.0 PL=0
MOVL C01714 V=800.0 PL=0
MOVL C01715 V=800.0 PL=0
MOVL C01716 V=800.0 PL=0
MOVL C01717 V=800.0 PL=0
MOVL C01718 V=800.0 PL=0
MOVL C01719 V=800.0 PL=0
MOVL C01720 V=800.0 PL=0
MOVL C01721 V=800.0 PL=0
MOVL C01722 V=800.0 PL=0
MOVL C01723 V=800.0 PL=0
MOVL C01724 V=800.0 PL=0
MOVL C01725 V=800.0 PL=0
MOVL C01726 V=800.0 PL=0
MOVL C01727 V=800.0 PL=0
MOVL C01728 V=800.0 PL=0
MOVL C01729 V=800.0 PL=0
MOVL C01730 V=800.0 PL=0
MOVL C01731 V=800.0 PL=0
MOVL C01732 V=800.0 PL=0
MOVL C01733 V=800.0 PL=0
MOVL C01734 V=800.0 PL=0
MOVL C01735 V=800.0 PL=0
MOVL C01736 V=800.0 PL=0
MOVL C01737 V=800.0 PL=0
MOVL C01738 V=800.0 PL=0
MOVL C01739 V=800.0 PL=0
MOVL C01740 V=800.0 PL=0
MOVL C01741 V=800.0 PL=0
MOVL C01742 V=800.0 PL=0
MOVL C01743 V=800.0 PL=0
MOVL C01744 V=800.0 PL=0
MOVL C01745 V=800.0 PL=0
MOVL C01746 V=800.0 PL=0
MOVL C01747 V=800.0 PL=0
MOVL C01748 V=800.0 PL=0
MOVL C01749 V=800.0 PL=0
MOVL C01750 V=800.0 PL=0
MOVL C01751 V=800.0 PL=0
MOVL C01752 V=800.0 PL=0
MOVL C01753 V=800.0 PL=0
MOVL C01754 V=800.0 PL=0
MOVL C01755 V=800.0 PL=0
MOVL C01756 V=800.0 PL=0
MOVL C01757 V=800.0 PL=0
MOVL C01758 V=800.0 PL=0
MOVL C01759 V=800.0 PL=0
MOVL C01760 V=800.0 PL=0
MOVL C01761 V=800.0 PL=0
MOVL C01762 V=800.0 PL=0
MOVL C01763 V=800.0 PL=0
MOVL C01764 V=800.0 PL=0
MOVL C01765 V=800.0 PL=0
MOVL C01766 V=800.0 PL=0
MOVL C01767 V=800.0 PL=0
MOVL C01768 V=800.0 PL=0
MOVL C01769 V=800.0 PL=0
MOVL C01770 V=800.0 PL=0
MOVL C01771 V=800.0 PL=0
MOVL C01772 V=800.0 PL=0
MOVL C01773 V=800.0 PL=0
MOVL C01774 V=800.0 PL=0
MOVL C01775 V=800.0 PL=0
MOVL C01776 V=800.0 PL=0
MOVL C01777 V=800.0 PL=0
MOVL C01778 V=800.0 PL=0
MOVL C01779 V=800.0 PL=0
MOVL C01780 V=800.0 PL=0
MOVL C01781 V=800.0 PL=0
MOVL C01782 V=800.0 PL=0
MOVL C01783 V=800.0 PL=0
MOVL C01784 V=800.0 PL=0
MOVL C01785 V=800.0 PL=0
MOVL C01786 V=800.0 PL=0
MOVL C01787 V=800.0 PL=0
MOVL C01788 V=800.0 PL=0
MOVL C01789 V=800.0 PL=0
MOVL C01790 V=800.0 PL=0
MOVL C01791 V=800.0 PL=0
MOVL C01792 V=800.0 PL=0
MOVL C01793 V=800.0 PL=0
MOVL C01794 V=800.0 PL=0
MOVL C01795 V=800.0 PL=0
MOVL C01796 V=800.0 PL=0
MOVL C01797 V=800.0 PL=0
MOVL C01798 V=800.0 PL=0
MOVL C01799 V=800.0 PL=0
MOVL C01800 V=800.0 PL=0
MOVL C01801 V=800.0 PL=0
MOVL C01802 V=800.0 PL=0
MOVL C01803 V=800.0 PL=0
MOVL C01804 V=800.0 PL=0
MOVL C01805 V=800.0 PL=0
MOVL C01806 V=800.0 PL=0
MOVL C01807 V=800.0 PL=0
MOVL C01808 V=800.0 PL=0
MOVL C01809 V=800.0 PL=0
MOVL C01810 V=800.0 PL=0
MOVL C01811 V=800.0 PL=0
MOVL C01812 V=800.0 PL=0
MOVL C01813 V=800.0 PL=0
MOVL C01814 V=800.0 PL=0
MOVL C01815 V=800.0 PL=0
MOVL C01816 V=800.0 PL=0
MOVL C01817 V=800.0 PL=0
MOVL C01818 V=800.0 PL=0
MOVL C01819 V=800.0 PL=0
MOVL C01820 V=800.0 PL=0
MOVL C01821 V=800.0 PL=0
MOVL C01822 V=800.0 PL=0
MOVL C01823 V=800.0 PL=0
MOVL C01824 V=800.0 PL=0
MOVL C01825 V=800.0 PL=0
MOVL C01826 V=800.0 PL=0
MOVL C01827 V=800.0 PL=0
MOVL C01828 V=800.0 PL=0
MOVL C01829 V=800.0 PL=0
MOVL C01830 V=800.0 PL=0
MOVL C01831 V=800.0 PL=0
MOVL C01832 V=800.0 PL=0
MOVL C01833 V=800.0 PL=0
MOVL C01834 V=800.0 PL=0
MOVL C01835 V=800.0 PL=0
MOVL C01836 V=800.0 PL=0
MOVL C01837 V=800.0 PL=0
MOVL C01838 V=800.0 PL=0
MOVL C01839 V=800.0 PL=0
MOVL C01840 V=800.0 PL=0
MOVL C01841 V=800.0 PL=0
MOVL C01842 V=800.0 PL=0
MOVL C01843 V=800.0 PL=0
MOVL C01844 V=800.0 PL=0
MOVL C01845 V=800.0 PL=0
MOVL C01846 V=800.0 PL=0
MOVL C01847 V=800.0 PL=0
MOVL C01848 V=800.0 PL=0
MOVL C01849 V=800.0 PL=0
MOVL C01850 V=800.0 PL=0
MOVL C01851 V=800.0 PL=0
MOVL C01852 V=800.0 PL=0
MOVL C01853 V=800.0 PL=0
MOVL C01854 V=800.0 PL=0
MOVL C01855 V=800.0 PL=0
MOVL C01856 V=800.0 PL=0
MOVL C01857 V=800.0 PL=0
MOVL C01858 V=800.0 PL=0
MOVL C01859 V=800.0 PL=0
MOVL C01860 V=800.0 PL=0
MOVL C01861 V=800.0 PL=0
MOVL C01862 V=800.0 PL=0
MOVL C01863 V=800.0 PL=0
MOVL C01864 V=800.0 PL=0
MOVL C01865 V=800.0 PL=0
MOVL C01866 V=800.0 PL=0
MOVL C01867 V=800.0 PL=0
MOVL C01868 V=800.0 PL=0
MOVL C01869 V=800.0 PL=0
MOVL C01870 V=800.0 PL=0
MOVL C01871 V=800.0 PL=0
MOVL C01872 V=800.0 PL=0
MOVL C01873 V=800.0 PL=0
MOVL C01874 V=800.0 PL=0
MOVL C01875 V=800.0 PL=0
MOVL C01876 V=800.0 PL=0
MOVL C01877 V=800.0 PL=0
MOVL C01878 V=800.0 PL=0
MOVL C01879 V=800.0 PL=0
MOVL C01880 V=800.0 PL=0
MOVL C01881 V=800.0 PL=0
MOVL C01882 V=800.0 PL=0
MOVL C01883 V=800.0 PL=0
MOVL C01884 V=800.0 PL=0
MOVL C01885 V=800.0 PL=0
MOVL C01886 V=800.0 PL=0
MOVL C01887 V=800.0 PL=0
MOVL C01888 V=800.0 PL=0
MOVL C01889 V=800.0 PL=0
MOVL C01890 V=800.0 PL=0
MOVL C01891 V=800.0 PL=0
MOVL C01892 V=800.0 PL=0
MOVL C01893 V=800.0 PL=0
MOVL C01894 V=800.0 PL=0
MOVL C01895 V=800.0 PL=0
MOVL C01896 V=800.0 PL=0
MOVL C01897 V=800.0 PL=0
MOVL C01898 V=800.0 PL=0
MOVL C01899 V=800.0 PL=0
MOVL C01900 V=800.0 PL=0
MOVL C01901 V=800.0 PL=0
MOVL C01902 V=800.0 PL=0
MOVL C01903 V=800.0 PL=0
MOVL C01904 V=800.0 PL=0
MOVL C01905 V=800.0 PL=0
MOVL C01906 V=800.0 PL=0
MOVL C01907 V=800.0 PL=0
MOVL C01908 V=800.0 PL=0
MOVL C01909 V=800.0 PL=0
MOVL C01910 V=800.0 PL=0
MOVL C01911 V=800.0 PL=0
MOVL C01912 V=800.0 PL=0
MOVL C01913 V=800.0 PL=0
MOVL C01914 V=800.0 PL=0
MOVL C01915 V=800.0 PL=0
MOVL C01916 V=800.0 PL=0
MOVL C01917 V=800.0 PL=0
MOVL C01918 V=800.0 PL=0
MOVL C01919 V=800.0 PL=0
MOVL C01920 V=800.0 PL=0
MOVL C01921 V=800.0 PL=0
MOVL C01922 V=800.0 PL=0
MOVL C01923 V=800.0 PL=0
MOVL C01924 V=800.0 PL=0
MOVL C01925 V=800.0 PL=0
MOVL C01926 V=800.0 PL=0
MOVL C01927 V=800.0 PL=0
MOVL C01928 V=800.0 PL=0
MOVL C01929 V=800.0 PL=0
MOVL C01930 V=800.0 PL=0
MOVL C01931 V=800.0 PL=0
MOVL C01932 V=800.0 PL=0
MOVL C01933 V=800.0 PL=0
MOVL C01934 V=800.0 PL=0
MOVL C01935 V=800.0 PL=0
MOVL C01936 V=800.0 PL=0
MOVL C01937 V=800.0 PL=0
MOVL C01938 V=800.0 PL=0
MOVL C01939 V=800.0 PL=0
MOVL C01940 V=800.0 PL=0
MOVL C01941 V=800.0 PL=0
MOVL C01942 V=800.0 PL=0
MOVL C01943 V=800.0 PL=0
MOVL C01944 V=800.0 PL=0
MOVL C01945 V=800.0 PL=0
MOVL C01946 V=800.0 PL=0
MOVL C01947 V=800.0 PL=0
MOVL C01948 V=800.0 PL=0
MOVL C01949 V=800.0 PL=0
MOVL C01950 V=800.0 PL=0
MOVL C01951 V=800.0 PL=0
MOVL C01952 V=800.0 PL=0
MOVL C01953 V=800.0 PL=0
MOVL C01954 V=800.0 PL=0
MOVL C01955 V=800.0 PL=0
MOVL C01956 V=800.0 PL=0
MOVL C01957 V=800.0 PL=0
MOVL C01958 V=800.0 PL=0
MOVL C01959 V=800.0 PL=0
MOVL C01960 V=800.0 PL=0
MOVL C01961 V=800.0 PL=0
MOVL C01962 V=800.0 PL=0
MOVL C01963 V=800.0 PL=0
MOVL C01964 V=800.0 PL=0
MOVL C01965 V=800.0 PL=0
MOVL C01966 V=800.0 PL=0
MOVL C01967 V=800.0 PL=0
MOVL C01968 V=800.0 PL=0
MOVL C01969 V=800.0 PL=0
MOVL C01970 V=800.0 PL=0
MOVL C01971 V=800.0 PL=0
MOVL C01972 V=800.0 PL=0
MOVL C01973 V=800.0 PL=0
MOVL C01974 V=800.0 PL=0
MOVL C01975 V=800.0 PL=0
MOVL C01976 V=800.0 PL=0
MOVL C01977 V=800.0 PL=0
MOVL C01978 V=800.0 PL=0
MOVL C01979 V=800.0 PL=0
MOVL C01980 V=800.0 PL=0
MOVL C01981 V=800.0 PL=0
MOVL C01982 V=800.0 PL=0
MOVL C01983 V=800.0 PL=0
MOVL C01984 V=800.0 PL=0
MOVL C01985 V=800.0 PL=0
MOVL C01986 V=800.0 PL=0
MOVL C01987 V=800.0 PL=0
MOVL C01988 V=800.0 PL=0
MOVL C01989 V=800.0 PL=0
MOVL C01990 V=800.0 PL=0
MOVL C01991 V=800.0 PL=0
MOVL C01992 V=800.0 PL=0
MOVL C01993 V=800.0 PL=0
MOVL C01994 V=800.0 PL=0
MOVL C01995 V=800.0 PL=0
MOVL C01996 V=800.0 PL=0
MOVL C01997 V=800.0 PL=0
MOVL C01998 V=800.0 PL=0
MOVL C01999 V=800.0 PL=0
MOVL C02000 V=800.0 PL=0
MOVL C02001 V=800.0 PL=0
MOVL C02002 V=800.0 PL=0
MOVL C02003 V=800.0 PL=0
MOVL C02004 V=800.0 PL=0
MOVL C02005 V=800.0 PL=0
MOVL C02006 V=800.0 PL=0
MOVL C02007 V=800.0 PL=0
MOVL C02008 V=800.0 PL=0
MOVL C02009 V=800.0 PL=0
MOVL C02010 V=800.0 PL=0
MOVL C02011 V=800.0 PL=0
MOVL C02012 V=800.0 PL=0
MOVL C02013 V=800.0 PL=0
MOVL C02014 V=800.0 PL=0
MOVL C02015 V=800.0 PL=0
MOVL C02016 V=800.0 PL=0
MOVL C02017 V=800.0 PL=0
MOVL C02018 V=800.0 PL=0
MOVL C02019 V=800.0 PL=0
MOVL C02020 V=800.0 PL=0
MOVL C02021 V=800.0 PL=0
MOVL C02022 V=800.0 PL=0
MOVL C02023 V=800.0 PL=0
MOVL C02024 V=800.0 PL=0
MOVL C02025 V=800.0 PL=0
MOVL C02026 V=800.0 PL=0
MOVL C02027 V=800.0 PL=0
MOVL C02028 V=800.0 PL=0
MOVL C02029 V=800.0 PL=0
MOVL C02030 V=800.0 PL=0
MOVL C02031 V=800.0 PL=0
MOVL C02032 V=800.0 PL=0
MOVL C02033 V=800.0 PL=0
MOVL C02034 V=800.0 PL=0
MOVL C02035 V=800.0 PL=0
